# B&R Automation Studio project TD52 (part 95)

#### VibMonEGInit.st
```iecst
(*******************************************************************************
VibMonEG: Vigration monitoring engine / generator (init)

This code is confidential AND proprietary to the INNIO Company.
It may NOT be used in any form, or reproduced in any manner, without the express
written permission of the INNIO Company.
Copyright, INNIO Company, 2021

- monitoring of vibration values incl. frequency bands
- determine max velocity and frequencay at maximum

Customized modifications: -
------------------------

History:
-------
V4.11.0	25-05-2021	Weitzer, 	generated
V4.11.1	04-02-2022	Schmid,		automatic PLC address detection
V4.11.2	20-01-2026	Bacci,		customized for DP29

Instructions FOR use:
--------------------
Sensor 1: Generator horizontal
Sensor 2: Generator vetical
Sensor 3: Engine horizontal
Sensor 4: Engine vetical

Outstandings:
------------

*******************************************************************************)

PROGRAM _INIT

//	(*========= DETERMINE POSITION OF X20CM4810 MODULE ==========*)
//	(* ********************************************************* *)
//	(*	reset variables											 *)
//	(* ********************************************************* *)
//	memset(ADR(sLabelInfo),	 	0, SIZEOF(sLabelInfo));
//
//	(* ********************************************************* *)
//	(*	get information about configured modules				 *)
//	(* ********************************************************* *)
//	xDiagCreateInfo_CM4810.enable	:= TRUE;
//	xDiagCreateInfo_CM4810.infoKind	:= asdiagCONFIGURED;
//	xDiagCreateInfo_CM4810();
//
//	IF (xDiagCreateInfo_CM4810.status = 0) THEN
//		iIdent 		:= xDiagCreateInfo_CM4810.ident;
//		iNrEntries	:= xDiagCreateInfo_CM4810.nrEntries;
//	END_IF;
//
//	(* ********************************************************* *)
//	(*	get module type of configured modules in Physical		 *)
//	(* ********************************************************* *)
//	FOR iIndex := 0 TO iNrEntries - 1 DO
//		xDiagGetStrInfo_CM4810.enable		:= TRUE;
//		xDiagGetStrInfo_CM4810.ident		:= iIdent;
//		xDiagGetStrInfo_CM4810.index		:= iIndex;
//		xDiagGetStrInfo_CM4810.infoCode		:= asdiagCONFIG_MODULE;
//		xDiagGetStrInfo_CM4810.pBuffer		:= ADR(sLabelInfo);
//		xDiagGetStrInfo_CM4810.bufferLen	:= SIZEOF(sLabelInfo) - 1;
//		xDiagGetStrInfo_CM4810();
//
//		IF (xDiagGetStrInfo_CM4810.status = 0) THEN
//		(* ********************************************************* *)
//		(*	get path of X20CM4810 module							 *)
//		(* ********************************************************* *)
//			IF FIND(sLabelInfo, 'X20CM4810') <> 0 THEN
//				xDiagGetStrInfo_CM4810.infoCode		:= asdiagPATH;
//				xDiagGetStrInfo_CM4810.pBuffer		:= ADR(sAddrInfo);
//				xDiagGetStrInfo_CM4810.bufferLen	:= SIZEOF(sAddrInfo) - 1;
//				xDiagGetStrInfo_CM4810();
//
//				IF (xDiagGetStrInfo_CM4810.status = 0) THEN
//					sCM4810Addr	:=	sAddrInfo;
//				END_IF;
//			END_IF;
//		END_IF;
//	END_FOR;
//
//	(* ********************************************************* *)
//	(*	free ressources of AsIODiag								 *)
//	(* ********************************************************* *)
//	xDiagDisposeInfo_CM4810.enable := TRUE;
//	xDiagDisposeInfo_CM4810.ident  := iIdent;
//	xDiagDisposeInfo_CM4810();
//	(*===========================================================*)

//  Prevent compiler warnings
	xDiagCreateInfo_CM4810.enable := FALSE;
	xDiagGetStrInfo_CM4810.enable := FALSE;
	xDiagDisposeInfo_CM4810.enable := FALSE;
	sLabelInfo;
	sAddrInfo;
	iIndex;
	iIdent;
	iNrEntries;

	//  PLC address of 1st X20CM4810 vibration module
	sCM4810Addr := 'IF3.ST33.IF1.ST2';

	(* init setting for CM4810 FUB *)
	xCM4810.paramMain.pModulePath			  := ADR(sCM4810Addr); 								(* set path to module *)

	xCM4810.enable							  := TRUE; 											(* enable FUB *)
	xCM4810.paramBufferUpload.nrArrayElements := SIZEOF(rData_x_Axis)/SIZEOF(rData_x_Axis[0]);	(* the length of the rData_x_Axis and rData_y_Axis arrays must be the same *)
	xCM4810.paramBufferUpload.pArrayXaxis	  := ADR(rData_x_Axis);								(* load buffer address x axis array *)
	xCM4810.paramBufferUpload.pArrayYaxis	  := ADR(rData_y_Axis);								(* load buffer address y axis array *)

	xCM4810.paramBufferUpload.moduleBuffer:= 66;    (* define module buffer for upload *)
	//moduleBuffer  Buffer description                        Signal source             Channel number   Number of values   y-axis unit    x-axis unit
	//    9         Buffered time signal (amplitude)          Raw acceleration signal      1                8192                [mg]       [seconds]
	//   11         Buffered time signal (amplitude)          Raw acceleration signal      2                8192                [mg]       [seconds]
	//   13         Buffered time signal (amplitude)          Raw acceleration signal      3                8192                [mg]       [seconds]
	//   15         Buffered time signal (amplitude)          Raw acceleration signal      4                8192                [mg]       [seconds]
	//   25         Buffered time signal (amplitude)          Envelope monitoring          1                8192                [mg]       [seconds]
	//   27         Buffered time signal (amplitude)          Envelope monitoring          2                8192                [mg]       [seconds]
	//   29         Buffered time signal (amplitude)          Envelope monitoring          3                8192                [mg]       [seconds]
	//   31         Buffered time signal (amplitude)          Envelope monitoring          4                8192                [mg]       [seconds]
	//   66         Spectrum buffered frequency (amplitude)   Raw velocity signal          1                4096                [mm/s]       [Hz]
	//   67         Spectrum buffered frequency (amplitude)   Raw acceleration signal      1                4096                [mg]         [Hz]
	//   70         Spectrum buffered frequency (amplitude)   Raw velocity signal          2                4096                [mm/s]       [Hz]
	//   71         Spectrum buffered frequency (amplitude)   Raw acceleration signal      2                4096                [mg]         [Hz]
	//   74         Spectrum buffered frequency (amplitude)   Raw velocity signal          3                4096                [mm/s]       [Hz]
	//   75         Spectrum buffered frequency (amplitude)   Raw acceleration signal      3                4096                [mg]         [Hz]
	//   78         Spectrum buffered frequency (amplitude)   Raw velocity signal          4                4096                [mm/s]       [Hz]
	//   79         Spectrum buffered frequency (amplitude)   Raw acceleration signal      4                4096                [mg]         [Hz]
	//   82         Spectrum buffered frequency (amplitude)   Envelope signal speed        1                4096                [mm/s]       [Hz]
	//   83         Spectrum buffered frequency (amplitude)   Envelope monitoring          1                4096                [mg]         [Hz]
	//   86         Spectrum buffered frequency (amplitude)   Envelope signal speed        2                4096                [mm/s]       [Hz]
	//   87         Spectrum buffered frequency (amplitude)   Envelope monitoring          2                4096                [mg]         [Hz]
	//   90         Spectrum buffered frequency (amplitude)   Envelope signal speed        3                4096                [mm/s]       [Hz]
	//   91         Spectrum buffered frequency (amplitude)   Envelope monitoring          3                4096                [mg]         [Hz]
	//   94         Spectrum buffered frequency (amplitude)   Envelope signal speed        4                4096                [mm/s]       [Hz]
	//   95         Spectrum buffered frequency (amplitude)   Envelope monitoring          4                4096                [mg]         [Hz]

	(* set sensor sensitivity *)
	rSensitivitySensor[1] := 100.0; (*mV/g*)
	rSensitivitySensor[2] := 100.0; (*mV/g*)
	rSensitivitySensor[3] := 100.0; (*mV/g*)
	rSensitivitySensor[4] := 100.0; (*mV/g*)

	(* Enable application of sensitivity on buffer *)
	xCM4810.paramMain.sensitivitySensor01:=rSensitivitySensor[1];
	xCM4810.paramMain.sensitivitySensor02:=rSensitivitySensor[2];
	xCM4810.paramMain.sensitivitySensor03:=rSensitivitySensor[3];
	xCM4810.paramMain.sensitivitySensor04:=rSensitivitySensor[4];

	(* initialize values *)
	tiCM4810_ReadBuffer := T#1m;
	iNum_VibSens		:= 1;

END_PROGRAM
```

#### VibMonEG.typ - Local data types
```iecst
TYPE
	stpCM4810_Enum :
		(
		stpInitDone,
		stpWaitStart,
		stpReqLockBuffer,
		stpUploadBuffer,
		stpReqUnlockBuffer,
		stpError
		);
END_TYPE
```

#### VibMonEG.var - Local variables
```iecst
VAR CONSTANT
	AxisArrayMaxIndex : UINT := 8191;
END_VAR
VAR
	bStartBufferUpload : BOOL := TRUE; (* in order to start the buffer upload, set to TRUE *)
	xCM4810 : vbioCtrlCM4810; (* FUB to read buffers of a CM4810 module *)
	stpCM4810 : stpCM4810_Enum; (* step of state machine *)
	rData_x_Axis : ARRAY[0..AxisArrayMaxIndex] OF REAL; (* array of x-axis values (time values [s] or frequency values [Hz]) *)
	rData_y_Axis : ARRAY[0..AxisArrayMaxIndex] OF REAL; (* array of y-axis values (vibration [mg] of [mm/s] values *)
	bWrite : BOOL;
	szWriteConfig : STRING[50];
	bRead : BOOL;
	szReadConfig : STRING[50];
	xAsIOAccWrite1 : AsIOAccWrite;
	xAsIOAccRead1 : AsIOAccRead;
	rSensitivitySensor : ARRAY[0..4] OF REAL;
	bGetFrequencyMax : BOOL;
	usCount : UINT;
	tiCM4810_ReadBuffer : TIME;
	xTON_ReadCycle : TON;
	iNum_VibSens : INT;
	rVel_VibSens_Band : ARRAY[0..32] OF REAL := [33(0)];
	rVel_VibSens : ARRAY[0..4] OF REAL := [5(0)];
	usMaxIndex : UINT;
	rVel_y_Axis_Max : REAL;
	bVibSens_Overflow : ARRAY[0..4] OF BOOL := [5(0)];
	bVibSens_BrokenWire : ARRAY[0..4] OF BOOL := [5(0)];
	ucWriteBandCnt : USINT := 0;
	rCenterBandOld1 : REAL := 0.0;
	rCenterBandOld2 : REAL := 0.0;
	rCenterBandOld3 : REAL := 0.0;
	rCenterBandOld4 : REAL := 0.0;
	rCenterBandOld5 : REAL := 0.0;
	rCenterBandOld6 : REAL := 0.0;
	rCenterBandOld7 : REAL := 0.0;
	rCenterBandOld8 : REAL := 0.0;
	rIdx_VibSens_BandWidtOld : REAL := 0.0;
END_VAR
VAR
	xDiagCreateInfo_CM4810 : DiagCreateInfo; (*Get number of configured modules*)
	xDiagGetStrInfo_CM4810 : DiagGetStrInfo; (*Get name of configured modules*)
	xDiagDisposeInfo_CM4810 : DiagDisposeInfo; (*Free ressources of AsIODiag*)
	sLabelInfo : STRING[50]; (*Includes label of configured module*)
	sAddrInfo : STRING[50]; (*Includes address of configured module*)
	iIndex : UDINT; (*Index of actual read module*)
	iIdent : UDINT; (*Ident from xDiagCreateInfo_CM4810*)
	iNrEntries : UDINT; (*Number of configured modules from xDiagCreateInfo_CM4810*)
	sCM4810Addr : STRING[50]; (*CM4810 IF PLC address string*)
END_VAR
```

### Program Logical/EngineGeneral/VibMon2EG (IEC, version 4.11.1) - Vibration monitoring eng & gen

#### VibMonEGCyclic.st - Init, cyclic, exit code
```iecst
(*******************************************************************************
VibMonEG: Vigration monitoring engine / generator (cyclic)

This code is confidential AND proprietary to the INNIO Company.
It may NOT be used in any form, or reproduced in any manner, without the express
written permission of the INNIO Company.
Copyright, INNIO Company, 2021

- monitoring of vibration values incl. frequency bands
- determine max velocity and frequencay at maximum

Customized modifications: -
------------------------

History:
-------
V4.11	25-05-2021	Weitzer, 	generated

Instructions FOR use:
--------------------
Sensor 1: Generator horizontal
Sensor 2: Generator vetical
Sensor 3: Engine horizontal
Sensor 4: Engine vetical

Outstandings:
------------

*******************************************************************************)

PROGRAM _CYCLIC

	(* code is only executed if function is activated by parameter and if system has completed the start up *)
	IF Para.bVibSens_Act AND IN_EG.tPB2MM.bSys_Run THEN

		(* mapping of data points from 4 vibration sensors *)
		FOR usCount := 0 TO 3 DO

			(* check if vibraton sensore wire break detected and engine speed is below start limit *)
			IF bVibSens_BrokenWire[usCount+1] OR IN_EG.rN_EngAct < Para.rN_EngStart_LimHi THEN
				(* vibration sensor live RMS values [mm/s]*)
				MM2VIS.rVel_VibSens[usCount+5] := 0;
				(* vibration sensor live frequency band [mm/s] *)
				MM2VIS.rVel_VibSens_Band1[usCount+5] := 0;
				MM2VIS.rVel_VibSens_Band2[usCount+5] := 0;
				MM2VIS.rVel_VibSens_Band3[usCount+5] := 0;
				MM2VIS.rVel_VibSens_Band4[usCount+5] := 0;
				MM2VIS.rVel_VibSens_Band5[usCount+5] := 0;
				MM2VIS.rVel_VibSens_Band6[usCount+5] := 0;
				MM2VIS.rVel_VibSens_Band7[usCount+5] := 0;
				MM2VIS.rVel_VibSens_Band8[usCount+5] := 0;
				(* vibration sensor max values *)
				MM2VIS.rVel_VibSens_Max[usCount+5] := 0;
				MM2VIS.rF_VibSens_Max[usCount+5]   := 0;
			(* check if no vibraton sensore overflow detected *)
			ELSIF NOT bVibSens_Overflow[usCount+1] THEN
				(* vibration sensor live RMS values [mm/s]*)
				MM2VIS.rVel_VibSens[usCount+5] := rVel_VibSens[usCount+1];					(* mapping directly from IO mapping, no HALIO used for vibration mesarurement *)
				(* vibration sensor live frequency band [mm/s] *)
				MM2VIS.rVel_VibSens_Band1[usCount+5] := rVel_VibSens_Band[usCount*8+1];		(* mapping directly from IO mapping, no HALIO used for vibration mesarurement *)
				MM2VIS.rVel_VibSens_Band2[usCount+5] := rVel_VibSens_Band[usCount*8+2];		(* mapping directly from IO mapping, no HALIO used for vibration mesarurement *)
				MM2VIS.rVel_VibSens_Band3[usCount+5] := rVel_VibSens_Band[usCount*8+3];		(* mapping directly from IO mapping, no HALIO used for vibration mesarurement *)
				MM2VIS.rVel_VibSens_Band4[usCount+5] := rVel_VibSens_Band[usCount*8+4];		(* mapping directly from IO mapping, no HALIO used for vibration mesarurement *)
				MM2VIS.rVel_VibSens_Band5[usCount+5] := rVel_VibSens_Band[usCount*8+5];		(* mapping directly from IO mapping, no HALIO used for vibration mesarurement *)
				MM2VIS.rVel_VibSens_Band6[usCount+5] := rVel_VibSens_Band[usCount*8+6];		(* mapping directly from IO mapping, no HALIO used for vibration mesarurement *)
				MM2VIS.rVel_VibSens_Band7[usCount+5] := rVel_VibSens_Band[usCount*8+7];		(* mapping directly from IO mapping, no HALIO used for vibration mesarurement *)
				MM2VIS.rVel_VibSens_Band8[usCount+5] := rVel_VibSens_Band[usCount*8+8];		(* mapping directly from IO mapping, no HALIO used for vibration mesarurement *)
			END_IF;

		END_FOR;

		(* read buffer data *)

		(* generate time interval for reading buffer *)
		xTON_ReadCycle(IN := NOT xTON_ReadCycle.Q, PT :=  tiCM4810_ReadBuffer);

		(* generate start reading trigger *)
		IF IN_EG.tEng_Run.Do AND stpCM4810 = stpWaitStart AND xTON_ReadCycle.Q THEN
			iNum_VibSens := iNum_VibSens + 1;
			IF iNum_VibSens > 4 THEN
				iNum_VibSens := 1;
			END_IF;
			bStartBufferUpload 					   := TRUE;
			xCM4810.paramBufferUpload.moduleBuffer := 66 + (iNum_VibSens-1) * 4;
		END_IF;

		(* state engine to read of data buffer *)

		CASE stpCM4810 OF
			//---------------------------------------------
			// wait for init done
			//---------------------------------------------
			stpInitDone:
				xCM4810.requestBufferLock := FALSE;
				xCM4810.uploadBuffer	  := FALSE;
				IF xCM4810.initDone AND xCM4810.moduleCfgUploadDone THEN
					stpCM4810 := stpWaitStart;
				END_IF;

			//---------------------------------------------
			// wait for start uplaod buffer
			//---------------------------------------------
			stpWaitStart:
				xCM4810.requestBufferLock := FALSE;
				xCM4810.uploadBuffer	  := FALSE;
				(* wait for start *)
				IF bStartBufferUpload THEN
					stpCM4810 := stpReqLockBuffer;
				END_IF;

			//---------------------------------------------
			// request lock buffer and wait until valid
			//---------------------------------------------
			stpReqLockBuffer:
				xCM4810.requestBufferLock := TRUE;
				bStartBufferUpload		  := FALSE; (* reset command start *)
				IF xCM4810.bufferLockValid THEN
					xCM4810.uploadBuffer := TRUE;
					stpCM4810			 := stpUploadBuffer;
				END_IF;

			//---------------------------------------------
			// upload buffer
			//---------------------------------------------
			stpUploadBuffer:
				IF xCM4810.bufferUploadDone THEN
					stpCM4810 := stpReqUnlockBuffer;
				END_IF;
				IF xCM4810.status <> ERR_FUB_BUSY AND xCM4810.status <> ERR_OK THEN
					stpCM4810 := stpError;
				END_IF

			//---------------------------------------------
			// unlock buffer and wait until valid
			//---------------------------------------------
			stpReqUnlockBuffer:
				xCM4810.requestBufferLock := FALSE;
				xCM4810.uploadBuffer	  := FALSE;
				IF NOT xCM4810.bufferLockValid THEN
					bGetFrequencyMax := TRUE;
					stpCM4810		 := stpWaitStart;
				END_IF;

			//---------------------------------------------
			// error
			//---------------------------------------------
			stpError:
			// no action!

		END_CASE;

		xCM4810.paramMain.pModulePath			  := ADR(sCM4810Addr);
		xCM4810.paramBufferUpload.pArrayXaxis	  := ADR(rData_x_Axis);
		xCM4810.paramBufferUpload.pArrayYaxis	  := ADR(rData_y_Axis);

		xCM4810(); (* call FUB exactly once per cycle *)

		(* get value & frequency max *)

		IF bGetFrequencyMax THEN

			MM2VIS.rF_VibSens_Max[iNum_VibSens+4]   := 0.0;		(* reset x(y max) max *)
			rVel_y_Axis_Max := 0.0;										(* reset y max *)
			usMaxIndex := 0;
			FOR usCount := 1 TO AxisArrayMaxIndex DO
				(* Upper limit for max value search at 500 Hz *)
				IF rData_x_Axis[usCount] > 500.0 THEN
					EXIT;
				END_IF
				(*find max signal value *)
				IF rData_y_Axis[usCount] > rVel_y_Axis_Max THEN
					rVel_y_Axis_Max := rData_y_Axis[usCount];		(* max virbration value *)
					MM2VIS.rF_VibSens_Max[iNum_VibSens+4]   := rData_x_Axis[usCount];		(* frequency at max virbration value *)
					usMaxIndex := usCount;
				END_IF
			END_FOR;

			(* correction of buffer value *)
			IF usMaxIndex > 1 AND usMaxIndex < (AxisArrayMaxIndex-2) THEN
				MM2VIS.rVel_VibSens_Max[iNum_VibSens+4] := 2.0/SQRT(3.0/2.0)*SQRT(0.5*(EXPT(rData_y_Axis[usMaxIndex-2],2)+EXPT(rData_y_Axis[usMaxIndex-1],2)+EXPT(rData_y_Axis[usMaxIndex],2)+EXPT(rData_y_Axis[usMaxIndex+1],2)+EXPT(rData_y_Axis[usMaxIndex+2],2)));
			ELSE
				MM2VIS.rVel_VibSens_Max[iNum_VibSens+4] := 0.0;
			END_IF;

			bGetFrequencyMax := FALSE;
		END_IF;

		(* calculate and display center frequency at the HMI *)

//		MM2VIS.rF_VibSens_CenterBand1 := Para.rN_EngNom/60.0*Para.rIdx_VibSens_BandOrder1;
//		MM2VIS.rF_VibSens_CenterBand2 := Para.rN_EngNom/60.0*Para.rIdx_VibSens_BandOrder2;
//		MM2VIS.rF_VibSens_CenterBand3 := Para.rN_EngNom/60.0*Para.rIdx_VibSens_BandOrder3;
//		MM2VIS.rF_VibSens_CenterBand4 := Para.rN_EngNom/60.0*Para.rIdx_VibSens_BandOrder4;
//		MM2VIS.rF_VibSens_CenterBand5 := Para.rN_EngNom/60.0*Para.rIdx_VibSens_BandOrder5;
//		MM2VIS.rF_VibSens_CenterBand6 := Para.rN_EngNom/60.0*Para.rIdx_VibSens_BandOrder6;
//		MM2VIS.rF_VibSens_CenterBand7 := Para.rN_EngNom/60.0*Para.rIdx_VibSens_BandOrder7;
//		MM2VIS.rF_VibSens_CenterBand8 := Para.rN_EngNom/60.0*Para.rIdx_VibSens_BandOrder8;

		(* check if band upper and lower frequency limit has to be set *)

		IF NOT bWrite THEN

			IF ucWriteBandCnt = 0 THEN

				IF Para.rIdx_VibSens_BandWidth <> rIdx_VibSens_BandWidtOld THEN
					rIdx_VibSens_BandWidtOld := Para.rIdx_VibSens_BandWidth;
					rCenterBandOld1			 := 0.0;
					rCenterBandOld2			 := 0.0;
					rCenterBandOld3			 := 0.0;
					rCenterBandOld4			 := 0.0;
					rCenterBandOld5			 := 0.0;
					rCenterBandOld6			 := 0.0;
					rCenterBandOld7			 := 0.0;
					rCenterBandOld8			 := 0.0;
				ELSIF MM2VIS.rF_VibSens_CenterBand1 <> rCenterBandOld1 THEN
					rCenterBandOld1 := MM2VIS.rF_VibSens_CenterBand1;
					ucWriteBandCnt  := 1;
				ELSIF MM2VIS.rF_VibSens_CenterBand2 <> rCenterBandOld2 THEN
					rCenterBandOld2 := MM2VIS.rF_VibSens_CenterBand2;
					ucWriteBandCnt  := 9;
				ELSIF MM2VIS.rF_VibSens_CenterBand3 <> rCenterBandOld3 THEN
					rCenterBandOld3 := MM2VIS.rF_VibSens_CenterBand3;
					ucWriteBandCnt  := 17;
				ELSIF MM2VIS.rF_VibSens_CenterBand4 <> rCenterBandOld4 THEN
					rCenterBandOld4 := MM2VIS.rF_VibSens_CenterBand4;
					ucWriteBandCnt  := 25;
				ELSIF MM2VIS.rF_VibSens_CenterBand5 <> rCenterBandOld5 THEN
					rCenterBandOld5 := MM2VIS.rF_VibSens_CenterBand5;
					ucWriteBandCnt  := 33;
				ELSIF MM2VIS.rF_VibSens_CenterBand6 <> rCenterBandOld6 THEN
					rCenterBandOld6 := MM2VIS.rF_VibSens_CenterBand6;
					ucWriteBandCnt  := 41;
				ELSIF MM2VIS.rF_VibSens_CenterBand7 <> rCenterBandOld7 THEN
					rCenterBandOld7 := MM2VIS.rF_VibSens_CenterBand7;
					ucWriteBandCnt  := 49;
				ELSIF MM2VIS.rF_VibSens_CenterBand8 <> rCenterBandOld8 THEN
					rCenterBandOld8 := MM2VIS.rF_VibSens_CenterBand8;
					ucWriteBandCnt  := 57;
				END_IF;

			END_IF;

			(* writing of the single band limit registers *)
			CASE ucWriteBandCnt OF

				(* Band 1 - Sensor 1 *)
				1:  bWrite		 		 := TRUE;
					szWriteConfig		 := 'FrequencyBand01LowerFrequency';
					xAsIOAccWrite1.value := LIMIT(1,REAL_TO_UDINT(4.0*(MM2VIS.rF_VibSens_CenterBand1 - Para.rIdx_VibSens_BandWidth/2)),40000);
					ucWriteBandCnt		 := 2;
				2:  bWrite		 		 := TRUE;
					szWriteConfig		 := 'FrequencyBand01UpperFrequency';
					xAsIOAccWrite1.value := LIMIT(1,REAL_TO_UDINT(4.0*(MM2VIS.rF_VibSens_CenterBand1 + Para.rIdx_VibSens_BandWidth/2)),40000);
					ucWriteBandCnt		 := 3;
				(* Band 1 - Sensor 2 *)
				3:  bWrite		 		 := TRUE;
					szWriteConfig		 := 'FrequencyBand09LowerFrequency';
					xAsIOAccWrite1.value := LIMIT(1,REAL_TO_UDINT(4.0*(MM2VIS.rF_VibSens_CenterBand1 - Para.rIdx_VibSens_BandWidth/2)),40000);
					ucWriteBandCnt		 := 4;
				4:  bWrite		 		 := TRUE;
					szWriteConfig		 := 'FrequencyBand09UpperFrequency';
					xAsIOAccWrite1.value := LIMIT(1,REAL_TO_UDINT(4.0*(MM2VIS.rF_VibSens_CenterBand1 + Para.rIdx_VibSens_BandWidth/2)),40000);
					ucWriteBandCnt		 := 5;
				(* Band 1 - Sensor 3 *)
				5:  bWrite		 		 := TRUE;
					szWriteConfig		 := 'FrequencyBand17LowerFrequency';
					xAsIOAccWrite1.value := LIMIT(1,REAL_TO_UDINT(4.0*(MM2VIS.rF_VibSens_CenterBand1 - Para.rIdx_VibSens_BandWidth/2)),40000);
					ucWriteBandCnt		 := 6;
				6:  bWrite		 		 := TRUE;
					szWriteConfig		 := 'FrequencyBand17UpperFrequency';
					xAsIOAccWrite1.value := LIMIT(1,REAL_TO_UDINT(4.0*(MM2VIS.rF_VibSens_CenterBand1 + Para.rIdx_VibSens_BandWidth/2)),40000);
					ucWriteBandCnt		 := 7;
				(* Band 1 - Sensor 4 *)
				7:  bWrite		 		 := TRUE;
					szWriteConfig		 := 'FrequencyBand25LowerFrequency';
					xAsIOAccWrite1.value := LIMIT(1,REAL_TO_UDINT(4.0*(MM2VIS.rF_VibSens_CenterBand1 - Para.rIdx_VibSens_BandWidth/2)),40000);
					ucWriteBandCnt		 := 8;
				8:  bWrite		 		 := TRUE;
					szWriteConfig		 := 'FrequencyBand25UpperFrequency';
					xAsIOAccWrite1.value := LIMIT(1,REAL_TO_UDINT(4.0*(MM2VIS.rF_VibSens_CenterBand1 + Para.rIdx_VibSens_BandWidth/2)),40000);
					ucWriteBandCnt		 := 0;

					(* Band 2 - Sensor 1 *)
				9:  bWrite		 		 := TRUE;
					szWriteConfig		 := 'FrequencyBand02LowerFrequency';
					xAsIOAccWrite1.value := LIMIT(1,REAL_TO_UDINT(4.0*(MM2VIS.rF_VibSens_CenterBand2 - Para.rIdx_VibSens_BandWidth/2)),40000);
					ucWriteBandCnt		 := 10;
				10: bWrite		 		 := TRUE;
					szWriteConfig		 := 'FrequencyBand02UpperFrequency';
					xAsIOAccWrite1.value := LIMIT(1,REAL_TO_UDINT(4.0*(MM2VIS.rF_VibSens_CenterBand2 + Para.rIdx_VibSens_BandWidth/2)),40000);
					ucWriteBandCnt		 := 11;
					(* Band 2 - Sensor 2 *)
				11: bWrite		 		 := TRUE;
					szWriteConfig		 := 'FrequencyBand10LowerFrequency';
					xAsIOAccWrite1.value := LIMIT(1,REAL_TO_UDINT(4.0*(MM2VIS.rF_VibSens_CenterBand2 - Para.rIdx_VibSens_BandWidth/2)),40000);
					ucWriteBandCnt		 := 12;
				12: bWrite		 		 := TRUE;
					szWriteConfig		 := 'FrequencyBand10UpperFrequency';
					xAsIOAccWrite1.value := LIMIT(1,REAL_TO_UDINT(4.0*(MM2VIS.rF_VibSens_CenterBand2 + Para.rIdx_VibSens_BandWidth/2)),40000);
					ucWriteBandCnt		 := 13;
					(* Band 2 - Sensor 3 *)
				13: bWrite		 		 := TRUE;
					szWriteConfig		 := 'FrequencyBand18LowerFrequency';
					xAsIOAccWrite1.value := LIMIT(1,REAL_TO_UDINT(4.0*(MM2VIS.rF_VibSens_CenterBand2 - Para.rIdx_VibSens_BandWidth/2)),40000);
					ucWriteBandCnt		 := 14;
				14: bWrite		 		 := TRUE;
					szWriteConfig		 := 'FrequencyBand18UpperFrequency';
					xAsIOAccWrite1.value := LIMIT(1,REAL_TO_UDINT(4.0*(MM2VIS.rF_VibSens_CenterBand2 + Para.rIdx_VibSens_BandWidth/2)),40000);
					ucWriteBandCnt		 := 15;
					(* Band 2 - Sensor 4 *)
				15: bWrite		 		 := TRUE;
					szWriteConfig		 := 'FrequencyBand26LowerFrequency';
					xAsIOAccWrite1.value := LIMIT(1,REAL_TO_UDINT(4.0*(MM2VIS.rF_VibSens_CenterBand2 - Para.rIdx_VibSens_BandWidth/2)),40000);
					ucWriteBandCnt		 := 16;
				16: bWrite		 		 := TRUE;
					szWriteConfig		 := 'FrequencyBand26UpperFrequency';
					xAsIOAccWrite1.value := LIMIT(1,REAL_TO_UDINT(4.0*(MM2VIS.rF_VibSens_CenterBand2 + Para.rIdx_VibSens_BandWidth/2)),40000);
					ucWriteBandCnt		 := 0;

					(* Band 3 - Sensor 1 *)
				17: bWrite		 		 := TRUE;
					szWriteConfig		 := 'FrequencyBand03LowerFrequency';
					xAsIOAccWrite1.value := LIMIT(1,REAL_TO_UDINT(4.0*(MM2VIS.rF_VibSens_CenterBand3 - Para.rIdx_VibSens_BandWidth/2)),40000);
					ucWriteBandCnt		 := 18;
				18: bWrite		 		 := TRUE;
					szWriteConfig		 := 'FrequencyBand03UpperFrequency';
					xAsIOAccWrite1.value := LIMIT(1,REAL_TO_UDINT(4.0*(MM2VIS.rF_VibSens_CenterBand3 + Para.rIdx_VibSens_BandWidth/2)),40000);
					ucWriteBandCnt		 := 19;
					(* Band 3 - Sensor 2 *)
				19: bWrite		 		 := TRUE;
					szWriteConfig		 := 'FrequencyBand11LowerFrequency';
					xAsIOAccWrite1.value := LIMIT(1,REAL_TO_UDINT(4.0*(MM2VIS.rF_VibSens_CenterBand3 - Para.rIdx_VibSens_BandWidth/2)),40000);
					ucWriteBandCnt		 := 20;
				20: bWrite		 		 := TRUE;
					szWriteConfig		 := 'FrequencyBand11UpperFrequency';
					xAsIOAccWrite1.value := LIMIT(1,REAL_TO_UDINT(4.0*(MM2VIS.rF_VibSens_CenterBand3 + Para.rIdx_VibSens_BandWidth/2)),40000);
					ucWriteBandCnt		 := 21;
					(* Band 3 - Sensor 3 *)
				21: bWrite		 		 := TRUE;
					szWriteConfig		 := 'FrequencyBand19LowerFrequency';
					xAsIOAccWrite1.value := LIMIT(1,REAL_TO_UDINT(4.0*(MM2VIS.rF_VibSens_CenterBand3 - Para.rIdx_VibSens_BandWidth/2)),40000);
					ucWriteBandCnt		 := 22;
				22: bWrite		 		 := TRUE;
					szWriteConfig		 := 'FrequencyBand19UpperFrequency';
					xAsIOAccWrite1.value := LIMIT(1,REAL_TO_UDINT(4.0*(MM2VIS.rF_VibSens_CenterBand3 + Para.rIdx_VibSens_BandWidth/2)),40000);
					ucWriteBandCnt		 := 23;
					(* Band 3 - Sensor 4 *)
				23: bWrite		 		 := TRUE;
					szWriteConfig		 := 'FrequencyBand27LowerFrequency';
					xAsIOAccWrite1.value := LIMIT(1,REAL_TO_UDINT(4.0*(MM2VIS.rF_VibSens_CenterBand3 - Para.rIdx_VibSens_BandWidth/2)),40000);
					ucWriteBandCnt		 := 24;
				24: bWrite		 		 := TRUE;
					szWriteConfig		 := 'FrequencyBand27UpperFrequency';
					xAsIOAccWrite1.value := LIMIT(1,REAL_TO_UDINT(4.0*(MM2VIS.rF_VibSens_CenterBand3 + Para.rIdx_VibSens_BandWidth/2)),40000);
					ucWriteBandCnt		 := 0;

					(* Band 4 - Sensor 1 *)
				25: bWrite		 		 := TRUE;
					szWriteConfig		 := 'FrequencyBand04LowerFrequency';
					xAsIOAccWrite1.value := LIMIT(1,REAL_TO_UDINT(4.0*(MM2VIS.rF_VibSens_CenterBand4 - Para.rIdx_VibSens_BandWidth/2)),40000);
					ucWriteBandCnt		 := 26;
				26: bWrite		 		 := TRUE;
					szWriteConfig		 := 'FrequencyBand04UpperFrequency';
					xAsIOAccWrite1.value := LIMIT(1,REAL_TO_UDINT(4.0*(MM2VIS.rF_VibSens_CenterBand4 + Para.rIdx_VibSens_BandWidth/2)),40000);
					ucWriteBandCnt		 := 27;
					(* Band 4 - Sensor 2 *)
				27: bWrite		 		 := TRUE;
					szWriteConfig		 := 'FrequencyBand12LowerFrequency';
					xAsIOAccWrite1.value := LIMIT(1,REAL_TO_UDINT(4.0*(MM2VIS.rF_VibSens_CenterBand4 - Para.rIdx_VibSens_BandWidth/2)),40000);
					ucWriteBandCnt		 := 28;
				28: bWrite		 		 := TRUE;
					szWriteConfig		 := 'FrequencyBand12UpperFrequency';
					xAsIOAccWrite1.value := LIMIT(1,REAL_TO_UDINT(4.0*(MM2VIS.rF_VibSens_CenterBand4 + Para.rIdx_VibSens_BandWidth/2)),40000);
					ucWriteBandCnt		 := 29;
					(* Band 4 - Sensor 3 *)
				29: bWrite		 		 := TRUE;
					szWriteConfig		 := 'FrequencyBand20LowerFrequency';
					xAsIOAccWrite1.value := LIMIT(1,REAL_TO_UDINT(4.0*(MM2VIS.rF_VibSens_CenterBand4 - Para.rIdx_VibSens_BandWidth/2)),40000);
					ucWriteBandCnt		 := 30;
				30: bWrite		 		 := TRUE;
					szWriteConfig		 := 'FrequencyBand20UpperFrequency';
					xAsIOAccWrite1.value := LIMIT(1,REAL_TO_UDINT(4.0*(MM2VIS.rF_VibSens_CenterBand4 + Para.rIdx_VibSens_BandWidth/2)),40000);
					ucWriteBandCnt		 := 31;
					(* Band 4 - Sensor 4 *)
				31: bWrite		 		 := TRUE;
					szWriteConfig		 := 'FrequencyBand28LowerFrequency';
					xAsIOAccWrite1.value := LIMIT(1,REAL_TO_UDINT(4.0*(MM2VIS.rF_VibSens_CenterBand4 - Para.rIdx_VibSens_BandWidth/2)),40000);
					ucWriteBandCnt		 := 32;
				32: bWrite		 		 := TRUE;
					szWriteConfig		 := 'FrequencyBand28UpperFrequency';
					xAsIOAccWrite1.value := LIMIT(1,REAL_TO_UDINT(4.0*(MM2VIS.rF_VibSens_CenterBand4 + Para.rIdx_VibSens_BandWidth/2)),40000);
					ucWriteBandCnt		 := 0;

					(* Band 5 - Sensor 1 *)
				33: bWrite		 		 := TRUE;
					szWriteConfig		 := 'FrequencyBand05LowerFrequency';
					xAsIOAccWrite1.value := LIMIT(1,REAL_TO_UDINT(4.0*(MM2VIS.rF_VibSens_CenterBand5 - Para.rIdx_VibSens_BandWidth/2)),40000);
					ucWriteBandCnt		 := 34;
				34: bWrite		 		 := TRUE;
					szWriteConfig		 := 'FrequencyBand05UpperFrequency';
					xAsIOAccWrite1.value := LIMIT(1,REAL_TO_UDINT(4.0*(MM2VIS.rF_VibSens_CenterBand5 + Para.rIdx_VibSens_BandWidth/2)),40000);
					ucWriteBandCnt		 := 35;
					(* Band 5 - Sensor 2 *)
				35: bWrite		 		 := TRUE;
					szWriteConfig		 := 'FrequencyBand13LowerFrequency';
					xAsIOAccWrite1.value := LIMIT(1,REAL_TO_UDINT(4.0*(MM2VIS.rF_VibSens_CenterBand5 - Para.rIdx_VibSens_BandWidth/2)),40000);
					ucWriteBandCnt		 := 36;
				36: bWrite		 		 := TRUE;
					szWriteConfig		 := 'FrequencyBand13UpperFrequency';
					xAsIOAccWrite1.value := LIMIT(1,REAL_TO_UDINT(4.0*(MM2VIS.rF_VibSens_CenterBand5 + Para.rIdx_VibSens_BandWidth/2)),40000);
					ucWriteBandCnt		 := 37;
					(* Band 5 - Sensor 3 *)
				37: bWrite		 		 := TRUE;
					szWriteConfig		 := 'FrequencyBand21LowerFrequency';
					xAsIOAccWrite1.value := LIMIT(1,REAL_TO_UDINT(4.0*(MM2VIS.rF_VibSens_CenterBand5 - Para.rIdx_VibSens_BandWidth/2)),40000);
					ucWriteBandCnt		 := 38;
				38: bWrite		 		 := TRUE;
					szWriteConfig		 := 'FrequencyBand21UpperFrequency';
					xAsIOAccWrite1.value := LIMIT(1,REAL_TO_UDINT(4.0*(MM2VIS.rF_VibSens_CenterBand5 + Para.rIdx_VibSens_BandWidth/2)),40000);
					ucWriteBandCnt		 := 39;
					(* Band 5 - Sensor 4 *)
				39: bWrite		 		 := TRUE;
					szWriteConfig		 := 'FrequencyBand29LowerFrequency';
					xAsIOAccWrite1.value := LIMIT(1,REAL_TO_UDINT(4.0*(MM2VIS.rF_VibSens_CenterBand5 - Para.rIdx_VibSens_BandWidth/2)),40000);
					ucWriteBandCnt		 := 40;
				40: bWrite		 		 := TRUE;
					szWriteConfig		 := 'FrequencyBand29UpperFrequency';
					xAsIOAccWrite1.value := LIMIT(1,REAL_TO_UDINT(4.0*(MM2VIS.rF_VibSens_CenterBand5 + Para.rIdx_VibSens_BandWidth/2)),40000);
					ucWriteBandCnt		 := 0;

					(* Band 6 - Sensor 1 *)
				41: bWrite		 		 := TRUE;
					szWriteConfig		 := 'FrequencyBand06LowerFrequency';
					xAsIOAccWrite1.value := LIMIT(1,REAL_TO_UDINT(4.0*(MM2VIS.rF_VibSens_CenterBand6 - Para.rIdx_VibSens_BandWidth/2)),40000);
					ucWriteBandCnt		 := 42;
				42: bWrite		 		 := TRUE;
					szWriteConfig		 := 'FrequencyBand06UpperFrequency';
					xAsIOAccWrite1.value := LIMIT(1,REAL_TO_UDINT(4.0*(MM2VIS.rF_VibSens_CenterBand6 + Para.rIdx_VibSens_BandWidth/2)),40000);
					ucWriteBandCnt		 := 43;
					(* Band 6 - Sensor 2 *)
				43: bWrite		 		 := TRUE;
					szWriteConfig		 := 'FrequencyBand14LowerFrequency';
					xAsIOAccWrite1.value := LIMIT(1,REAL_TO_UDINT(4.0*(MM2VIS.rF_VibSens_CenterBand6 - Para.rIdx_VibSens_BandWidth/2)),40000);
					ucWriteBandCnt		 := 44;
				44: bWrite		 		 := TRUE;
					szWriteConfig		 := 'FrequencyBand14UpperFrequency';
					xAsIOAccWrite1.value := LIMIT(1,REAL_TO_UDINT(4.0*(MM2VIS.rF_VibSens_CenterBand6 + Para.rIdx_VibSens_BandWidth/2)),40000);
					ucWriteBandCnt		 := 45;
					(* Band 6 - Sensor 3 *)
				45: bWrite		 		 := TRUE;
					szWriteConfig		 := 'FrequencyBand22LowerFrequency';
					xAsIOAccWrite1.value := LIMIT(1,REAL_TO_UDINT(4.0*(MM2VIS.rF_VibSens_CenterBand6 - Para.rIdx_VibSens_BandWidth/2)),40000);
					ucWriteBandCnt		 := 46;
				46: bWrite		 		 := TRUE;
					szWriteConfig		 := 'FrequencyBand22UpperFrequency';
					xAsIOAccWrite1.value := LIMIT(1,REAL_TO_UDINT(4.0*(MM2VIS.rF_VibSens_CenterBand6 + Para.rIdx_VibSens_BandWidth/2)),40000);
					ucWriteBandCnt		 := 47;
					(* Band 6 - Sensor 4 *)
				47: bWrite		 		 := TRUE;
					szWriteConfig		 := 'FrequencyBand30LowerFrequency';
					xAsIOAccWrite1.value := LIMIT(1,REAL_TO_UDINT(4.0*(MM2VIS.rF_VibSens_CenterBand6 - Para.rIdx_VibSens_BandWidth/2)),40000);
					ucWriteBandCnt		 := 48;
				48: bWrite		 		 := TRUE;
					szWriteConfig		 := 'FrequencyBand30UpperFrequency';
					xAsIOAccWrite1.value := LIMIT(1,REAL_TO_UDINT(4.0*(MM2VIS.rF_VibSens_CenterBand6 + Para.rIdx_VibSens_BandWidth/2)),40000);
					ucWriteBandCnt		 := 0;

					(* Band 7 - Sensor 1 *)
				49: bWrite		 		 := TRUE;
					szWriteConfig		 := 'FrequencyBand07LowerFrequency';
					xAsIOAccWrite1.value := LIMIT(1,REAL_TO_UDINT(4.0*(MM2VIS.rF_VibSens_CenterBand7 - Para.rIdx_VibSens_BandWidth/2)),40000);
					ucWriteBandCnt		 := 50;
				50: bWrite		 		 := TRUE;
					szWriteConfig		 := 'FrequencyBand07UpperFrequency';
					xAsIOAccWrite1.value := LIMIT(1,REAL_TO_UDINT(4.0*(MM2VIS.rF_VibSens_CenterBand7 + Para.rIdx_VibSens_BandWidth/2)),40000);
					ucWriteBandCnt		 := 51;
					(* Band 7 - Sensor 2 *)
				51: bWrite		 		 := TRUE;
					szWriteConfig		 := 'FrequencyBand15LowerFrequency';
					xAsIOAccWrite1.value := LIMIT(1,REAL_TO_UDINT(4.0*(MM2VIS.rF_VibSens_CenterBand7 - Para.rIdx_VibSens_BandWidth/2)),40000);
					ucWriteBandCnt		 := 52;
				52: bWrite		 		 := TRUE;
					szWriteConfig		 := 'FrequencyBand15UpperFrequency';
					xAsIOAccWrite1.value := LIMIT(1,REAL_TO_UDINT(4.0*(MM2VIS.rF_VibSens_CenterBand7 + Para.rIdx_VibSens_BandWidth/2)),40000);
					ucWriteBandCnt		 := 53;
					(* Band 7 - Sensor 3 *)
				53: bWrite		 		 := TRUE;
					szWriteConfig		 := 'FrequencyBand23LowerFrequency';
					xAsIOAccWrite1.value := LIMIT(1,REAL_TO_UDINT(4.0*(MM2VIS.rF_VibSens_CenterBand7 - Para.rIdx_VibSens_BandWidth/2)),40000);
					ucWriteBandCnt		 := 54;
				54: bWrite		 		 := TRUE;
					szWriteConfig		 := 'FrequencyBand23UpperFrequency';
					xAsIOAccWrite1.value := LIMIT(1,REAL_TO_UDINT(4.0*(MM2VIS.rF_VibSens_CenterBand7 + Para.rIdx_VibSens_BandWidth/2)),40000);
					ucWriteBandCnt		 := 55;
					(* Band 7 - Sensor 4 *)
				55: bWrite		 		 := TRUE;
					szWriteConfig		 := 'FrequencyBand31LowerFrequency';
					xAsIOAccWrite1.value := LIMIT(1,REAL_TO_UDINT(4.0*(MM2VIS.rF_VibSens_CenterBand7 - Para.rIdx_VibSens_BandWidth/2)),40000);
					ucWriteBandCnt		 := 56;
				56: bWrite		 		 := TRUE;
					szWriteConfig		 := 'FrequencyBand31UpperFrequency';
					xAsIOAccWrite1.value := LIMIT(1,REAL_TO_UDINT(4.0*(MM2VIS.rF_VibSens_CenterBand7 + Para.rIdx_VibSens_BandWidth/2)),40000);
					ucWriteBandCnt		 := 0;

					(* Band 8 - Sensor 1 *)
				57: bWrite		 		 := TRUE;
					szWriteConfig		 := 'FrequencyBand08LowerFrequency';
					xAsIOAccWrite1.value := LIMIT(1,REAL_TO_UDINT(4.0*(MM2VIS.rF_VibSens_CenterBand8 - Para.rIdx_VibSens_BandWidth/2)),40000);
					ucWriteBandCnt		 := 58;
				58: bWrite		 		 := TRUE;
					szWriteConfig		 := 'FrequencyBand08UpperFrequency';
					xAsIOAccWrite1.value := LIMIT(1,REAL_TO_UDINT(4.0*(MM2VIS.rF_VibSens_CenterBand8 + Para.rIdx_VibSens_BandWidth/2)),40000);
					ucWriteBandCnt		 := 59;
					(* Band 8 - Sensor 2 *)
				59: bWrite		 		 := TRUE;
					szWriteConfig		 := 'FrequencyBand16LowerFrequency';
					xAsIOAccWrite1.value := LIMIT(1,REAL_TO_UDINT(4.0*(MM2VIS.rF_VibSens_CenterBand8 - Para.rIdx_VibSens_BandWidth/2)),40000);
					ucWriteBandCnt		 := 60;
				60: bWrite		 		 := TRUE;
					szWriteConfig		 := 'FrequencyBand16UpperFrequency';
					xAsIOAccWrite1.value := LIMIT(1,REAL_TO_UDINT(4.0*(MM2VIS.rF_VibSens_CenterBand8 + Para.rIdx_VibSens_BandWidth/2)),40000);
					ucWriteBandCnt		 := 61;
					(* Band 8 - Sensor 3 *)
				61: bWrite		 		 := TRUE;
					szWriteConfig		 := 'FrequencyBand24LowerFrequency';
					xAsIOAccWrite1.value := LIMIT(1,REAL_TO_UDINT(4.0*(MM2VIS.rF_VibSens_CenterBand8 - Para.rIdx_VibSens_BandWidth/2)),40000);
					ucWriteBandCnt		 := 62;
				62: bWrite		 		 := TRUE;
					szWriteConfig		 := 'FrequencyBand24UpperFrequency';
					xAsIOAccWrite1.value := LIMIT(1,REAL_TO_UDINT(4.0*(MM2VIS.rF_VibSens_CenterBand8 + Para.rIdx_VibSens_BandWidth/2)),40000);
					ucWriteBandCnt		 := 63;
					(* Band 8 - Sensor 4 *)
				63: bWrite		 		 := TRUE;
					szWriteConfig		 := 'FrequencyBand32LowerFrequency';
					xAsIOAccWrite1.value := LIMIT(1,REAL_TO_UDINT(4.0*(MM2VIS.rF_VibSens_CenterBand8 - Para.rIdx_VibSens_BandWidth/2)),40000);
					ucWriteBandCnt		 := 64;
				64: bWrite		 		 := TRUE;
					szWriteConfig		 := 'FrequencyBand32UpperFrequency';
					xAsIOAccWrite1.value := LIMIT(1,REAL_TO_UDINT(4.0*(MM2VIS.rF_VibSens_CenterBand8 + Para.rIdx_VibSens_BandWidth/2)),40000);
					ucWriteBandCnt		 := 0;

			END_CASE;

		END_IF;

		(* read & write X204810 registers *)

		(* write band configuration and miscellaneous values *)
		IF bWrite THEN														(* set bWrite to TRUE to write a register on the CM48810 X20 module *)
			xAsIOAccWrite1.enable	    := TRUE;
			xAsIOAccWrite1.pDeviceName  := xCM4810.paramMain.pModulePath;
//			xAsIOAccWrite1.value	    := 0;								(* set value to write at this attribute of the function block *)
			xAsIOAccWrite1.pChannelName	:= ADR(szWriteConfig);				(* set name of register to write at string pv szWriteConfig *)
			xAsIOAccWrite1();

			IF xAsIOAccWrite1.status = 0 THEN
				bWrite := FALSE;
			END_IF;
		END_IF;

		(* read miscellaneous values *)
		IF bRead THEN														(* set bRead to TRUE to read a register from the CM48810 X20 module *)
			xAsIOAccRead1.enable	   := TRUE;
			xAsIOAccRead1.pDeviceName  := xCM4810.paramMain.pModulePath;
//			xAsIOAccRead1.value;											(* here the read valure can be found *)
			xAsIOAccRead1.pChannelName := ADR(szReadConfig);				(* set name of register to read at string pv szReadConfig *)
			xAsIOAccRead1();

			IF xAsIOAccRead1.status = 0 THEN
				bRead := FALSE;
			END_IF;
		END_IF;

	END_IF;

END_PROGRAM
```

#### VibMonEGInit.st
```iecst
(*******************************************************************************
VibMonEG: Vigration monitoring engine / generator (init)

This code is confidential AND proprietary to the INNIO Company.
It may NOT be used in any form, or reproduced in any manner, without the express
written permission of the INNIO Company.
Copyright, INNIO Company, 2023

- monitoring of vibration values incl. frequency bands
- determine max velocity and frequencay at maximum

Customized modifications: -
------------------------

History:
-------
V4.11.1	20-01-2026	Bacci,	customized for DP29, generated from VibMonEG 4.11.1

Instructions FOR use:
--------------------
Sensor 1: Generator horizontal
Sensor 2: Generator vetical
Sensor 3: Engine horizontal
Sensor 4: Engine vetical

Outstandings:
------------

*******************************************************************************)

PROGRAM _INIT

//	(*========= DETERMINE POSITION OF X20CM4810 MODULE ==========*)
//	(* ********************************************************* *)
//	(*	reset variables											 *)
//	(* ********************************************************* *)
//	memset(ADR(sLabelInfo),	 	0, SIZEOF(sLabelInfo));
//
//	(* ********************************************************* *)
//	(*	get information about configured modules				 *)
//	(* ********************************************************* *)
//	xDiagCreateInfo_CM4810.enable	:= TRUE;
//	xDiagCreateInfo_CM4810.infoKind	:= asdiagCONFIGURED;
//	xDiagCreateInfo_CM4810();
//
//	IF (xDiagCreateInfo_CM4810.status = 0) THEN
//		iIdent 		:= xDiagCreateInfo_CM4810.ident;
//		iNrEntries	:= xDiagCreateInfo_CM4810.nrEntries;
//	END_IF;
//
//	(* ********************************************************* *)
//	(*	get module type of configured modules in Physical		 *)
//	(* ********************************************************* *)
//	FOR iIndex := 0 TO iNrEntries - 1 DO
//		xDiagGetStrInfo_CM4810.enable		:= TRUE;
//		xDiagGetStrInfo_CM4810.ident		:= iIdent;
//		xDiagGetStrInfo_CM4810.index		:= iIndex;
//		xDiagGetStrInfo_CM4810.infoCode		:= asdiagCONFIG_MODULE;
//		xDiagGetStrInfo_CM4810.pBuffer		:= ADR(sLabelInfo);
//		xDiagGetStrInfo_CM4810.bufferLen	:= SIZEOF(sLabelInfo) - 1;
//		xDiagGetStrInfo_CM4810();
//
//		IF (xDiagGetStrInfo_CM4810.status = 0) THEN
//		(* ********************************************************* *)
//		(*	get path of X20CM4810 module							 *)
//		(* ********************************************************* *)
//			IF FIND(sLabelInfo, 'X20CM4810') <> 0 THEN
//				xDiagGetStrInfo_CM4810.infoCode		:= asdiagPATH;
//				xDiagGetStrInfo_CM4810.pBuffer		:= ADR(sAddrInfo);
//				xDiagGetStrInfo_CM4810.bufferLen	:= SIZEOF(sAddrInfo) - 1;
//				xDiagGetStrInfo_CM4810();
//
//				IF (xDiagGetStrInfo_CM4810.status = 0) THEN
//					sCM4810Addr	:=	sAddrInfo;
//				END_IF;
//			END_IF;
//		END_IF;
//	END_FOR;
//
//	(* ********************************************************* *)
//	(*	free ressources of AsIODiag								 *)
//	(* ********************************************************* *)
//	xDiagDisposeInfo_CM4810.enable := TRUE;
//	xDiagDisposeInfo_CM4810.ident  := iIdent;
//	xDiagDisposeInfo_CM4810();
//	(*===========================================================*)

//  Prevent compiler warninga
	xDiagCreateInfo_CM4810.enable := FALSE;
	xDiagGetStrInfo_CM4810.enable := FALSE;
	xDiagDisposeInfo_CM4810.enable := FALSE;
	sLabelInfo;
	sAddrInfo;
	iIndex;
	iIdent;
	iNrEntries;

//  PLC address of 2nd X20CM4810 vibration module
	sCM4810Addr := 'IF3.ST33.IF1.ST3';

	(* init setting for CM4810 FUB *)
	xCM4810.paramMain.pModulePath			  := ADR(sCM4810Addr); 								(* set path to module *)

	xCM4810.enable							  := TRUE; 											(* enable FUB *)
	xCM4810.paramBufferUpload.nrArrayElements := SIZEOF(rData_x_Axis)/SIZEOF(rData_x_Axis[0]);	(* the length of the rData_x_Axis and rData_y_Axis arrays must be the same *)
	xCM4810.paramBufferUpload.pArrayXaxis	  := ADR(rData_x_Axis);								(* load buffer address x axis array *)
	xCM4810.paramBufferUpload.pArrayYaxis	  := ADR(rData_y_Axis);								(* load buffer address y axis array *)

	xCM4810.paramBufferUpload.moduleBuffer:= 66;    (* define module buffer for upload *)
	//moduleBuffer  Buffer description                        Signal source             Channel number   Number of values   y-axis unit    x-axis unit
	//    9         Buffered time signal (amplitude)          Raw acceleration signal      1                8192                [mg]       [seconds]
	//   11         Buffered time signal (amplitude)          Raw acceleration signal      2                8192                [mg]       [seconds]
	//   13         Buffered time signal (amplitude)          Raw acceleration signal      3                8192                [mg]       [seconds]
	//   15         Buffered time signal (amplitude)          Raw acceleration signal      4                8192                [mg]       [seconds]
	//   25         Buffered time signal (amplitude)          Envelope monitoring          1                8192                [mg]       [seconds]
	//   27         Buffered time signal (amplitude)          Envelope monitoring          2                8192                [mg]       [seconds]
	//   29         Buffered time signal (amplitude)          Envelope monitoring          3                8192                [mg]       [seconds]
	//   31         Buffered time signal (amplitude)          Envelope monitoring          4                8192                [mg]       [seconds]
	//   66         Spectrum buffered frequency (amplitude)   Raw velocity signal          1                4096                [mm/s]       [Hz]
	//   67         Spectrum buffered frequency (amplitude)   Raw acceleration signal      1                4096                [mg]         [Hz]
	//   70         Spectrum buffered frequency (amplitude)   Raw velocity signal          2                4096                [mm/s]       [Hz]
	//   71         Spectrum buffered frequency (amplitude)   Raw acceleration signal      2                4096                [mg]         [Hz]
	//   74         Spectrum buffered frequency (amplitude)   Raw velocity signal          3                4096                [mm/s]       [Hz]
	//   75         Spectrum buffered frequency (amplitude)   Raw acceleration signal      3                4096                [mg]         [Hz]
	//   78         Spectrum buffered frequency (amplitude)   Raw velocity signal          4                4096                [mm/s]       [Hz]
	//   79         Spectrum buffered frequency (amplitude)   Raw acceleration signal      4                4096                [mg]         [Hz]
	//   82         Spectrum buffered frequency (amplitude)   Envelope signal speed        1                4096                [mm/s]       [Hz]
	//   83         Spectrum buffered frequency (amplitude)   Envelope monitoring          1                4096                [mg]         [Hz]
	//   86         Spectrum buffered frequency (amplitude)   Envelope signal speed        2                4096                [mm/s]       [Hz]
	//   87         Spectrum buffered frequency (amplitude)   Envelope monitoring          2                4096                [mg]         [Hz]
	//   90         Spectrum buffered frequency (amplitude)   Envelope signal speed        3                4096                [mm/s]       [Hz]
	//   91         Spectrum buffered frequency (amplitude)   Envelope monitoring          3                4096                [mg]         [Hz]
	//   94         Spectrum buffered frequency (amplitude)   Envelope signal speed        4                4096                [mm/s]       [Hz]
	//   95         Spectrum buffered frequency (amplitude)   Envelope monitoring          4                4096                [mg]         [Hz]

	(* set sensor sensitivity *)
	rSensitivitySensor[1] := 100.0; (*mV/g*)
	rSensitivitySensor[2] := 100.0; (*mV/g*)
	rSensitivitySensor[3] := 100.0; (*mV/g*)
	rSensitivitySensor[4] := 100.0; (*mV/g*)

	(* Enable application of sensitivity on buffer *)
	xCM4810.paramMain.sensitivitySensor01:=rSensitivitySensor[1];
	xCM4810.paramMain.sensitivitySensor02:=rSensitivitySensor[2];
	xCM4810.paramMain.sensitivitySensor03:=rSensitivitySensor[3];
	xCM4810.paramMain.sensitivitySensor04:=rSensitivitySensor[4];

	(* initialize values *)
	tiCM4810_ReadBuffer := T#1m;
	iNum_VibSens		:= 1;

END_PROGRAM
```

#### VibMonEG.typ - Local data types
```iecst
TYPE
	stpCM4810_Enum :
		(
		stpInitDone,
		stpWaitStart,
		stpReqLockBuffer,
		stpUploadBuffer,
		stpReqUnlockBuffer,
		stpError
		);
END_TYPE
```

#### VibMonEG.var - Local variables
```iecst
VAR CONSTANT
	AxisArrayMaxIndex : UINT := 8191;
END_VAR
VAR
	bStartBufferUpload : BOOL := TRUE; (* in order to start the buffer upload, set to TRUE *)
	xCM4810 : vbioCtrlCM4810; (* FUB to read buffers of a CM4810 module *)
	stpCM4810 : stpCM4810_Enum; (* step of state machine *)
	rData_x_Axis : ARRAY[0..AxisArrayMaxIndex] OF REAL; (* array of x-axis values (time values [s] or frequency values [Hz]) *)
	rData_y_Axis : ARRAY[0..AxisArrayMaxIndex] OF REAL; (* array of y-axis values (vibration [mg] of [mm/s] values *)
	bWrite : BOOL;
	szWriteConfig : STRING[50];
	bRead : BOOL;
	szReadConfig : STRING[50];
	xAsIOAccWrite1 : AsIOAccWrite;
	xAsIOAccRead1 : AsIOAccRead;
	rSensitivitySensor : ARRAY[0..4] OF REAL;
	bGetFrequencyMax : BOOL;
	usCount : UINT;
	tiCM4810_ReadBuffer : TIME;
	xTON_ReadCycle : TON;
	iNum_VibSens : INT;
	rVel_VibSens_Band : ARRAY[0..32] OF REAL := [33(0)];
	rVel_VibSens : ARRAY[0..4] OF REAL := [5(0)];
	usMaxIndex : UINT;
	rVel_y_Axis_Max : REAL;
	bVibSens_Overflow : ARRAY[0..4] OF BOOL := [5(0)];
	bVibSens_BrokenWire : ARRAY[0..4] OF BOOL := [5(0)];
	ucWriteBandCnt : USINT := 0;
	rCenterBandOld1 : REAL := 0.0;
	rCenterBandOld2 : REAL := 0.0;
	rCenterBandOld3 : REAL := 0.0;
	rCenterBandOld4 : REAL := 0.0;
	rCenterBandOld5 : REAL := 0.0;
	rCenterBandOld6 : REAL := 0.0;
	rCenterBandOld7 : REAL := 0.0;
	rCenterBandOld8 : REAL := 0.0;
	rIdx_VibSens_BandWidtOld : REAL := 0.0;
END_VAR
VAR
	xDiagCreateInfo_CM4810 : DiagCreateInfo; (*Get number of configured modules*)
	xDiagGetStrInfo_CM4810 : DiagGetStrInfo; (*Get name of configured modules*)
	xDiagDisposeInfo_CM4810 : DiagDisposeInfo; (*Free ressources of AsIODiag*)
	sLabelInfo : STRING[50]; (*Includes label of configured module*)
	sAddrInfo : STRING[50]; (*Includes address of configured module*)
	iIndex : UDINT; (*Index of actual read module*)
	iIdent : UDINT; (*Ident from xDiagCreateInfo_CM4810*)
	iNrEntries : UDINT; (*Number of configured modules from xDiagCreateInfo_CM4810*)
	sCM4810Addr : STRING[50]; (*CM4810 IF PLC address string*)
END_VAR
```

### Program Logical/EngineGeneral/VibMon3EG (IEC, version 4.11.1) - Vibration monitoring eng & gen

#### VibMonEGCyclic.st - Init, cyclic, exit code
```iecst
(*******************************************************************************
VibMonEG: Vigration monitoring engine / generator (cyclic)

This code is confidential AND proprietary to the INNIO Company.
It may NOT be used in any form, or reproduced in any manner, without the express
written permission of the INNIO Company.
Copyright, INNIO Company, 2021

- monitoring of vibration values incl. frequency bands
- determine max velocity and frequencay at maximum

Customized modifications: -
------------------------

History:
-------
V4.11	25-05-2021	Weitzer, 	generated

Instructions FOR use:
--------------------
Sensor 1: Generator horizontal
Sensor 2: Generator vetical
Sensor 3: Engine horizontal
Sensor 4: Engine vetical

Outstandings:
------------

*******************************************************************************)

PROGRAM _CYCLIC

	(* code is only executed if function is activated by parameter and if system has completed the start up *)
	IF Para.bVibSens_Act AND IN_EG.tPB2MM.bSys_Run THEN

		(* mapping of data points from 4 vibration sensors *)
		FOR usCount := 0 TO 3 DO

			(* check if vibraton sensore wire break detected and engine speed is below start limit *)
			IF bVibSens_BrokenWire[usCount+1] OR IN_EG.rN_EngAct < Para.rN_EngStart_LimHi THEN
				(* vibration sensor live RMS values [mm/s]*)
				MM2VIS.rVel_VibSens[usCount+9] := 0;
				(* vibration sensor live frequency band [mm/s] *)
				MM2VIS.rVel_VibSens_Band1[usCount+9] := 0;
				MM2VIS.rVel_VibSens_Band2[usCount+9] := 0;
				MM2VIS.rVel_VibSens_Band3[usCount+9] := 0;
				MM2VIS.rVel_VibSens_Band4[usCount+9] := 0;
				MM2VIS.rVel_VibSens_Band5[usCount+9] := 0;
				MM2VIS.rVel_VibSens_Band6[usCount+9] := 0;
				MM2VIS.rVel_VibSens_Band7[usCount+9] := 0;
				MM2VIS.rVel_VibSens_Band8[usCount+9] := 0;
				(* vibration sensor max values *)
				MM2VIS.rVel_VibSens_Max[usCount+9] := 0;
				MM2VIS.rF_VibSens_Max[usCount+9]   := 0;
			(* check if no vibraton sensore overflow detected *)
			ELSIF NOT bVibSens_Overflow[usCount+1] THEN
				(* vibration sensor live RMS values [mm/s]*)
				MM2VIS.rVel_VibSens[usCount+9] := rVel_VibSens[usCount+1];					(* mapping directly from IO mapping, no HALIO used for vibration mesarurement *)
				(* vibration sensor live frequency band [mm/s] *)
				MM2VIS.rVel_VibSens_Band1[usCount+9] := rVel_VibSens_Band[usCount*8+1];		(* mapping directly from IO mapping, no HALIO used for vibration mesarurement *)
				MM2VIS.rVel_VibSens_Band2[usCount+9] := rVel_VibSens_Band[usCount*8+2];		(* mapping directly from IO mapping, no HALIO used for vibration mesarurement *)
				MM2VIS.rVel_VibSens_Band3[usCount+9] := rVel_VibSens_Band[usCount*8+3];		(* mapping directly from IO mapping, no HALIO used for vibration mesarurement *)
				MM2VIS.rVel_VibSens_Band4[usCount+9] := rVel_VibSens_Band[usCount*8+4];		(* mapping directly from IO mapping, no HALIO used for vibration mesarurement *)
				MM2VIS.rVel_VibSens_Band5[usCount+9] := rVel_VibSens_Band[usCount*8+5];		(* mapping directly from IO mapping, no HALIO used for vibration mesarurement *)
				MM2VIS.rVel_VibSens_Band6[usCount+9] := rVel_VibSens_Band[usCount*8+6];		(* mapping directly from IO mapping, no HALIO used for vibration mesarurement *)
				MM2VIS.rVel_VibSens_Band7[usCount+9] := rVel_VibSens_Band[usCount*8+7];		(* mapping directly from IO mapping, no HALIO used for vibration mesarurement *)
				MM2VIS.rVel_VibSens_Band8[usCount+9] := rVel_VibSens_Band[usCount*8+8];		(* mapping directly from IO mapping, no HALIO used for vibration mesarurement *)
			END_IF;

		END_FOR;

		(* read buffer data *)

		(* generate time interval for reading buffer *)
		xTON_ReadCycle(IN := NOT xTON_ReadCycle.Q, PT :=  tiCM4810_ReadBuffer);

		(* generate start reading trigger *)
		IF IN_EG.tEng_Run.Do AND stpCM4810 = stpWaitStart AND xTON_ReadCycle.Q THEN
			iNum_VibSens := iNum_VibSens + 1;
			IF iNum_VibSens > 4 THEN
				iNum_VibSens := 1;
			END_IF;
			bStartBufferUpload 					   := TRUE;
			xCM4810.paramBufferUpload.moduleBuffer := 66 + (iNum_VibSens-1) * 4;
		END_IF;

		(* state engine to read of data buffer *)

		CASE stpCM4810 OF
			//---------------------------------------------
			// wait for init done
			//---------------------------------------------
			stpInitDone:
				xCM4810.requestBufferLock := FALSE;
				xCM4810.uploadBuffer	  := FALSE;
				IF xCM4810.initDone AND xCM4810.moduleCfgUploadDone THEN
					stpCM4810 := stpWaitStart;
				END_IF;

			//---------------------------------------------
			// wait for start uplaod buffer
			//---------------------------------------------
			stpWaitStart:
				xCM4810.requestBufferLock := FALSE;
				xCM4810.uploadBuffer	  := FALSE;
				(* wait for start *)
				IF bStartBufferUpload THEN
					stpCM4810 := stpReqLockBuffer;
				END_IF;

			//---------------------------------------------
			// request lock buffer and wait until valid
			//---------------------------------------------
			stpReqLockBuffer:
				xCM4810.requestBufferLock := TRUE;
				bStartBufferUpload		  := FALSE; (* reset command start *)
				IF xCM4810.bufferLockValid THEN
					xCM4810.uploadBuffer := TRUE;
					stpCM4810			 := stpUploadBuffer;
				END_IF;

			//---------------------------------------------
			// upload buffer
			//---------------------------------------------
			stpUploadBuffer:
				IF xCM4810.bufferUploadDone THEN
					stpCM4810 := stpReqUnlockBuffer;
				END_IF;
				IF xCM4810.status <> ERR_FUB_BUSY AND xCM4810.status <> ERR_OK THEN
					stpCM4810 := stpError;
				END_IF

			//---------------------------------------------
			// unlock buffer and wait until valid
			//---------------------------------------------
			stpReqUnlockBuffer:
				xCM4810.requestBufferLock := FALSE;
				xCM4810.uploadBuffer	  := FALSE;
				IF NOT xCM4810.bufferLockValid THEN
					bGetFrequencyMax := TRUE;
					stpCM4810		 := stpWaitStart;
				END_IF;

			//---------------------------------------------
			// error
			//---------------------------------------------
			stpError:
			// no action!

		END_CASE;

		xCM4810.paramMain.pModulePath			  := ADR(sCM4810Addr);
		xCM4810.paramBufferUpload.pArrayXaxis	  := ADR(rData_x_Axis);
		xCM4810.paramBufferUpload.pArrayYaxis	  := ADR(rData_y_Axis);

		xCM4810(); (* call FUB exactly once per cycle *)

		(* get value & frequency max *)

		IF bGetFrequencyMax THEN

			MM2VIS.rF_VibSens_Max[iNum_VibSens+8]   := 0.0;		(* reset x(y max) max *)
			rVel_y_Axis_Max := 0.0;										(* reset y max *)
			usMaxIndex := 0;
			FOR usCount := 1 TO AxisArrayMaxIndex DO
				(* Upper limit for max value search at 500 Hz *)
				IF rData_x_Axis[usCount] > 500.0 THEN
					EXIT;
				END_IF
				(*find max signal value *)
				IF rData_y_Axis[usCount] > rVel_y_Axis_Max THEN
					rVel_y_Axis_Max := rData_y_Axis[usCount];		(* max virbration value *)
					MM2VIS.rF_VibSens_Max[iNum_VibSens+8]   := rData_x_Axis[usCount];		(* frequency at max virbration value *)
					usMaxIndex := usCount;
				END_IF
			END_FOR;

			(* correction of buffer value *)
			IF usMaxIndex > 1 AND usMaxIndex < (AxisArrayMaxIndex-2) THEN
				MM2VIS.rVel_VibSens_Max[iNum_VibSens+8] := 2.0/SQRT(3.0/2.0)*SQRT(0.5*(EXPT(rData_y_Axis[usMaxIndex-2],2)+EXPT(rData_y_Axis[usMaxIndex-1],2)+EXPT(rData_y_Axis[usMaxIndex],2)+EXPT(rData_y_Axis[usMaxIndex+1],2)+EXPT(rData_y_Axis[usMaxIndex+2],2)));
			ELSE
				MM2VIS.rVel_VibSens_Max[iNum_VibSens+8] := 0.0;
			END_IF;

			bGetFrequencyMax := FALSE;
		END_IF;

		(* calculate and display center frequency at the HMI *)

//		MM2VIS.rF_VibSens_CenterBand1 := Para.rN_EngNom/60.0*Para.rIdx_VibSens_BandOrder1;
//		MM2VIS.rF_VibSens_CenterBand2 := Para.rN_EngNom/60.0*Para.rIdx_VibSens_BandOrder2;
//		MM2VIS.rF_VibSens_CenterBand3 := Para.rN_EngNom/60.0*Para.rIdx_VibSens_BandOrder3;
//		MM2VIS.rF_VibSens_CenterBand4 := Para.rN_EngNom/60.0*Para.rIdx_VibSens_BandOrder4;
//		MM2VIS.rF_VibSens_CenterBand5 := Para.rN_EngNom/60.0*Para.rIdx_VibSens_BandOrder5;
//		MM2VIS.rF_VibSens_CenterBand6 := Para.rN_EngNom/60.0*Para.rIdx_VibSens_BandOrder6;
//		MM2VIS.rF_VibSens_CenterBand7 := Para.rN_EngNom/60.0*Para.rIdx_VibSens_BandOrder7;
//		MM2VIS.rF_VibSens_CenterBand8 := Para.rN_EngNom/60.0*Para.rIdx_VibSens_BandOrder8;

		(* check if band upper and lower frequency limit has to be set *)

		IF NOT bWrite THEN

			IF ucWriteBandCnt = 0 THEN

				IF Para.rIdx_VibSens_BandWidth <> rIdx_VibSens_BandWidtOld THEN
					rIdx_VibSens_BandWidtOld := Para.rIdx_VibSens_BandWidth;
					rCenterBandOld1			 := 0.0;
					rCenterBandOld2			 := 0.0;
					rCenterBandOld3			 := 0.0;
					rCenterBandOld4			 := 0.0;
					rCenterBandOld5			 := 0.0;
					rCenterBandOld6			 := 0.0;
					rCenterBandOld7			 := 0.0;
					rCenterBandOld8			 := 0.0;
				ELSIF MM2VIS.rF_VibSens_CenterBand1 <> rCenterBandOld1 THEN
					rCenterBandOld1 := MM2VIS.rF_VibSens_CenterBand1;
					ucWriteBandCnt  := 1;
				ELSIF MM2VIS.rF_VibSens_CenterBand2 <> rCenterBandOld2 THEN
					rCenterBandOld2 := MM2VIS.rF_VibSens_CenterBand2;
					ucWriteBandCnt  := 9;
				ELSIF MM2VIS.rF_VibSens_CenterBand3 <> rCenterBandOld3 THEN
					rCenterBandOld3 := MM2VIS.rF_VibSens_CenterBand3;
					ucWriteBandCnt  := 17;
				ELSIF MM2VIS.rF_VibSens_CenterBand4 <> rCenterBandOld4 THEN
					rCenterBandOld4 := MM2VIS.rF_VibSens_CenterBand4;
					ucWriteBandCnt  := 25;
				ELSIF MM2VIS.rF_VibSens_CenterBand5 <> rCenterBandOld5 THEN
					rCenterBandOld5 := MM2VIS.rF_VibSens_CenterBand5;
					ucWriteBandCnt  := 33;
				ELSIF MM2VIS.rF_VibSens_CenterBand6 <> rCenterBandOld6 THEN
					rCenterBandOld6 := MM2VIS.rF_VibSens_CenterBand6;
					ucWriteBandCnt  := 41;
				ELSIF MM2VIS.rF_VibSens_CenterBand7 <> rCenterBandOld7 THEN
					rCenterBandOld7 := MM2VIS.rF_VibSens_CenterBand7;
					ucWriteBandCnt  := 49;
				ELSIF MM2VIS.rF_VibSens_CenterBand8 <> rCenterBandOld8 THEN
					rCenterBandOld8 := MM2VIS.rF_VibSens_CenterBand8;
					ucWriteBandCnt  := 57;
				END_IF;

			END_IF;

			(* writing of the single band limit registers *)
			CASE ucWriteBandCnt OF

				(* Band 1 - Sensor 1 *)
				1:  bWrite		 		 := TRUE;
					szWriteConfig		 := 'FrequencyBand01LowerFrequency';
					xAsIOAccWrite1.value := LIMIT(1,REAL_TO_UDINT(4.0*(MM2VIS.rF_VibSens_CenterBand1 - Para.rIdx_VibSens_BandWidth/2)),40000);
					ucWriteBandCnt		 := 2;
				2:  bWrite		 		 := TRUE;
					szWriteConfig		 := 'FrequencyBand01UpperFrequency';
					xAsIOAccWrite1.value := LIMIT(1,REAL_TO_UDINT(4.0*(MM2VIS.rF_VibSens_CenterBand1 + Para.rIdx_VibSens_BandWidth/2)),40000);
					ucWriteBandCnt		 := 3;
				(* Band 1 - Sensor 2 *)
				3:  bWrite		 		 := TRUE;
					szWriteConfig		 := 'FrequencyBand09LowerFrequency';
					xAsIOAccWrite1.value := LIMIT(1,REAL_TO_UDINT(4.0*(MM2VIS.rF_VibSens_CenterBand1 - Para.rIdx_VibSens_BandWidth/2)),40000);
					ucWriteBandCnt		 := 4;
				4:  bWrite		 		 := TRUE;
					szWriteConfig		 := 'FrequencyBand09UpperFrequency';
					xAsIOAccWrite1.value := LIMIT(1,REAL_TO_UDINT(4.0*(MM2VIS.rF_VibSens_CenterBand1 + Para.rIdx_VibSens_BandWidth/2)),40000);
					ucWriteBandCnt		 := 5;
				(* Band 1 - Sensor 3 *)
				5:  bWrite		 		 := TRUE;
					szWriteConfig		 := 'FrequencyBand17LowerFrequency';
					xAsIOAccWrite1.value := LIMIT(1,REAL_TO_UDINT(4.0*(MM2VIS.rF_VibSens_CenterBand1 - Para.rIdx_VibSens_BandWidth/2)),40000);
					ucWriteBandCnt		 := 6;
				6:  bWrite		 		 := TRUE;
					szWriteConfig		 := 'FrequencyBand17UpperFrequency';
					xAsIOAccWrite1.value := LIMIT(1,REAL_TO_UDINT(4.0*(MM2VIS.rF_VibSens_CenterBand1 + Para.rIdx_VibSens_BandWidth/2)),40000);
					ucWriteBandCnt		 := 7;
				(* Band 1 - Sensor 4 *)
				7:  bWrite		 		 := TRUE;
					szWriteConfig		 := 'FrequencyBand25LowerFrequency';
					xAsIOAccWrite1.value := LIMIT(1,REAL_TO_UDINT(4.0*(MM2VIS.rF_VibSens_CenterBand1 - Para.rIdx_VibSens_BandWidth/2)),40000);
					ucWriteBandCnt		 := 8;
				8:  bWrite		 		 := TRUE;
					szWriteConfig		 := 'FrequencyBand25UpperFrequency';
					xAsIOAccWrite1.value := LIMIT(1,REAL_TO_UDINT(4.0*(MM2VIS.rF_VibSens_CenterBand1 + Para.rIdx_VibSens_BandWidth/2)),40000);
					ucWriteBandCnt		 := 0;

					(* Band 2 - Sensor 1 *)
				9:  bWrite		 		 := TRUE;
					szWriteConfig		 := 'FrequencyBand02LowerFrequency';
					xAsIOAccWrite1.value := LIMIT(1,REAL_TO_UDINT(4.0*(MM2VIS.rF_VibSens_CenterBand2 - Para.rIdx_VibSens_BandWidth/2)),40000);
					ucWriteBandCnt		 := 10;
				10: bWrite		 		 := TRUE;
					szWriteConfig		 := 'FrequencyBand02UpperFrequency';
					xAsIOAccWrite1.value := LIMIT(1,REAL_TO_UDINT(4.0*(MM2VIS.rF_VibSens_CenterBand2 + Para.rIdx_VibSens_BandWidth/2)),40000);
					ucWriteBandCnt		 := 11;
					(* Band 2 - Sensor 2 *)
				11: bWrite		 		 := TRUE;
					szWriteConfig		 := 'FrequencyBand10LowerFrequency';
					xAsIOAccWrite1.value := LIMIT(1,REAL_TO_UDINT(4.0*(MM2VIS.rF_VibSens_CenterBand2 - Para.rIdx_VibSens_BandWidth/2)),40000);
					ucWriteBandCnt		 := 12;
				12: bWrite		 		 := TRUE;
					szWriteConfig		 := 'FrequencyBand10UpperFrequency';
					xAsIOAccWrite1.value := LIMIT(1,REAL_TO_UDINT(4.0*(MM2VIS.rF_VibSens_CenterBand2 + Para.rIdx_VibSens_BandWidth/2)),40000);
					ucWriteBandCnt		 := 13;
					(* Band 2 - Sensor 3 *)
				13: bWrite		 		 := TRUE;
					szWriteConfig		 := 'FrequencyBand18LowerFrequency';
					xAsIOAccWrite1.value := LIMIT(1,REAL_TO_UDINT(4.0*(MM2VIS.rF_VibSens_CenterBand2 - Para.rIdx_VibSens_BandWidth/2)),40000);
					ucWriteBandCnt		 := 14;
				14: bWrite		 		 := TRUE;
					szWriteConfig		 := 'FrequencyBand18UpperFrequency';
					xAsIOAccWrite1.value := LIMIT(1,REAL_TO_UDINT(4.0*(MM2VIS.rF_VibSens_CenterBand2 + Para.rIdx_VibSens_BandWidth/2)),40000);
					ucWriteBandCnt		 := 15;
					(* Band 2 - Sensor 4 *)
				15: bWrite		 		 := TRUE;
					szWriteConfig		 := 'FrequencyBand26LowerFrequency';
					xAsIOAccWrite1.value := LIMIT(1,REAL_TO_UDINT(4.0*(MM2VIS.rF_VibSens_CenterBand2 - Para.rIdx_VibSens_BandWidth/2)),40000);
					ucWriteBandCnt		 := 16;
				16: bWrite		 		 := TRUE;
					szWriteConfig		 := 'FrequencyBand26UpperFrequency';
					xAsIOAccWrite1.value := LIMIT(1,REAL_TO_UDINT(4.0*(MM2VIS.rF_VibSens_CenterBand2 + Para.rIdx_VibSens_BandWidth/2)),40000);
					ucWriteBandCnt		 := 0;

					(* Band 3 - Sensor 1 *)
				17: bWrite		 		 := TRUE;
					szWriteConfig		 := 'FrequencyBand03LowerFrequency';
					xAsIOAccWrite1.value := LIMIT(1,REAL_TO_UDINT(4.0*(MM2VIS.rF_VibSens_CenterBand3 - Para.rIdx_VibSens_BandWidth/2)),40000);
					ucWriteBandCnt		 := 18;
				18: bWrite		 		 := TRUE;
					szWriteConfig		 := 'FrequencyBand03UpperFrequency';
					xAsIOAccWrite1.value := LIMIT(1,REAL_TO_UDINT(4.0*(MM2VIS.rF_VibSens_CenterBand3 + Para.rIdx_VibSens_BandWidth/2)),40000);
					ucWriteBandCnt		 := 19;
					(* Band 3 - Sensor 2 *)
				19: bWrite		 		 := TRUE;
					szWriteConfig		 := 'FrequencyBand11LowerFrequency';
					xAsIOAccWrite1.value := LIMIT(1,REAL_TO_UDINT(4.0*(MM2VIS.rF_VibSens_CenterBand3 - Para.rIdx_VibSens_BandWidth/2)),40000);
					ucWriteBandCnt		 := 20;
				20: bWrite		 		 := TRUE;
					szWriteConfig		 := 'FrequencyBand11UpperFrequency';
					xAsIOAccWrite1.value := LIMIT(1,REAL_TO_UDINT(4.0*(MM2VIS.rF_VibSens_CenterBand3 + Para.rIdx_VibSens_BandWidth/2)),40000);
					ucWriteBandCnt		 := 21;
					(* Band 3 - Sensor 3 *)
				21: bWrite		 		 := TRUE;
					szWriteConfig		 := 'FrequencyBand19LowerFrequency';
					xAsIOAccWrite1.value := LIMIT(1,REAL_TO_UDINT(4.0*(MM2VIS.rF_VibSens_CenterBand3 - Para.rIdx_VibSens_BandWidth/2)),40000);
					ucWriteBandCnt		 := 22;
				22: bWrite		 		 := TRUE;
					szWriteConfig		 := 'FrequencyBand19UpperFrequency';
					xAsIOAccWrite1.value := LIMIT(1,REAL_TO_UDINT(4.0*(MM2VIS.rF_VibSens_CenterBand3 + Para.rIdx_VibSens_BandWidth/2)),40000);
					ucWriteBandCnt		 := 23;
					(* Band 3 - Sensor 4 *)
				23: bWrite		 		 := TRUE;
					szWriteConfig		 := 'FrequencyBand27LowerFrequency';
					xAsIOAccWrite1.value := LIMIT(1,REAL_TO_UDINT(4.0*(MM2VIS.rF_VibSens_CenterBand3 - Para.rIdx_VibSens_BandWidth/2)),40000);
					ucWriteBandCnt		 := 24;
				24: bWrite		 		 := TRUE;
					szWriteConfig		 := 'FrequencyBand27UpperFrequency';
					xAsIOAccWrite1.value := LIMIT(1,REAL_TO_UDINT(4.0*(MM2VIS.rF_VibSens_CenterBand3 + Para.rIdx_VibSens_BandWidth/2)),40000);
					ucWriteBandCnt		 := 0;

					(* Band 4 - Sensor 1 *)
				25: bWrite		 		 := TRUE;
					szWriteConfig		 := 'FrequencyBand04LowerFrequency';
					xAsIOAccWrite1.value := LIMIT(1,REAL_TO_UDINT(4.0*(MM2VIS.rF_VibSens_CenterBand4 - Para.rIdx_VibSens_BandWidth/2)),40000);
					ucWriteBandCnt		 := 26;
				26: bWrite		 		 := TRUE;
					szWriteConfig		 := 'FrequencyBand04UpperFrequency';
					xAsIOAccWrite1.value := LIMIT(1,REAL_TO_UDINT(4.0*(MM2VIS.rF_VibSens_CenterBand4 + Para.rIdx_VibSens_BandWidth/2)),40000);
					ucWriteBandCnt		 := 27;
					(* Band 4 - Sensor 2 *)
				27: bWrite		 		 := TRUE;
					szWriteConfig		 := 'FrequencyBand12LowerFrequency';
					xAsIOAccWrite1.value := LIMIT(1,REAL_TO_UDINT(4.0*(MM2VIS.rF_VibSens_CenterBand4 - Para.rIdx_VibSens_BandWidth/2)),40000);
					ucWriteBandCnt		 := 28;
				28: bWrite		 		 := TRUE;
					szWriteConfig		 := 'FrequencyBand12UpperFrequency';
					xAsIOAccWrite1.value := LIMIT(1,REAL_TO_UDINT(4.0*(MM2VIS.rF_VibSens_CenterBand4 + Para.rIdx_VibSens_BandWidth/2)),40000);
					ucWriteBandCnt		 := 29;
					(* Band 4 - Sensor 3 *)
				29: bWrite		 		 := TRUE;
					szWriteConfig		 := 'FrequencyBand20LowerFrequency';
					xAsIOAccWrite1.value := LIMIT(1,REAL_TO_UDINT(4.0*(MM2VIS.rF_VibSens_CenterBand4 - Para.rIdx_VibSens_BandWidth/2)),40000);
					ucWriteBandCnt		 := 30;
				30: bWrite		 		 := TRUE;
					szWriteConfig		 := 'FrequencyBand20UpperFrequency';
					xAsIOAccWrite1.value := LIMIT(1,REAL_TO_UDINT(4.0*(MM2VIS.rF_VibSens_CenterBand4 + Para.rIdx_VibSens_BandWidth/2)),40000);
					ucWriteBandCnt		 := 31;
					(* Band 4 - Sensor 4 *)
				31: bWrite		 		 := TRUE;
					szWriteConfig		 := 'FrequencyBand28LowerFrequency';
					xAsIOAccWrite1.value := LIMIT(1,REAL_TO_UDINT(4.0*(MM2VIS.rF_VibSens_CenterBand4 - Para.rIdx_VibSens_BandWidth/2)),40000);
					ucWriteBandCnt		 := 32;
				32: bWrite		 		 := TRUE;
					szWriteConfig		 := 'FrequencyBand28UpperFrequency';
					xAsIOAccWrite1.value := LIMIT(1,REAL_TO_UDINT(4.0*(MM2VIS.rF_VibSens_CenterBand4 + Para.rIdx_VibSens_BandWidth/2)),40000);
					ucWriteBandCnt		 := 0;

					(* Band 5 - Sensor 1 *)
				33: bWrite		 		 := TRUE;
					szWriteConfig		 := 'FrequencyBand05LowerFrequency';
					xAsIOAccWrite1.value := LIMIT(1,REAL_TO_UDINT(4.0*(MM2VIS.rF_VibSens_CenterBand5 - Para.rIdx_VibSens_BandWidth/2)),40000);
					ucWriteBandCnt		 := 34;
				34: bWrite		 		 := TRUE;
					szWriteConfig		 := 'FrequencyBand05UpperFrequency';
					xAsIOAccWrite1.value := LIMIT(1,REAL_TO_UDINT(4.0*(MM2VIS.rF_VibSens_CenterBand5 + Para.rIdx_VibSens_BandWidth/2)),40000);
					ucWriteBandCnt		 := 35;
					(* Band 5 - Sensor 2 *)
				35: bWrite		 		 := TRUE;
					szWriteConfig		 := 'FrequencyBand13LowerFrequency';
					xAsIOAccWrite1.value := LIMIT(1,REAL_TO_UDINT(4.0*(MM2VIS.rF_VibSens_CenterBand5 - Para.rIdx_VibSens_BandWidth/2)),40000);
					ucWriteBandCnt		 := 36;
				36: bWrite		 		 := TRUE;
					szWriteConfig		 := 'FrequencyBand13UpperFrequency';
					xAsIOAccWrite1.value := LIMIT(1,REAL_TO_UDINT(4.0*(MM2VIS.rF_VibSens_CenterBand5 + Para.rIdx_VibSens_BandWidth/2)),40000);
					ucWriteBandCnt		 := 37;
					(* Band 5 - Sensor 3 *)
				37: bWrite		 		 := TRUE;
					szWriteConfig		 := 'FrequencyBand21LowerFrequency';
					xAsIOAccWrite1.value := LIMIT(1,REAL_TO_UDINT(4.0*(MM2VIS.rF_VibSens_CenterBand5 - Para.rIdx_VibSens_BandWidth/2)),40000);
					ucWriteBandCnt		 := 38;
				38: bWrite		 		 := TRUE;
					szWriteConfig		 := 'FrequencyBand21UpperFrequency';
					xAsIOAccWrite1.value := LIMIT(1,REAL_TO_UDINT(4.0*(MM2VIS.rF_VibSens_CenterBand5 + Para.rIdx_VibSens_BandWidth/2)),40000);
					ucWriteBandCnt		 := 39;
					(* Band 5 - Sensor 4 *)
				39: bWrite		 		 := TRUE;
					szWriteConfig		 := 'FrequencyBand29LowerFrequency';
					xAsIOAccWrite1.value := LIMIT(1,REAL_TO_UDINT(4.0*(MM2VIS.rF_VibSens_CenterBand5 - Para.rIdx_VibSens_BandWidth/2)),40000);
					ucWriteBandCnt		 := 40;
				40: bWrite		 		 := TRUE;
					szWriteConfig		 := 'FrequencyBand29UpperFrequency';
					xAsIOAccWrite1.value := LIMIT(1,REAL_TO_UDINT(4.0*(MM2VIS.rF_VibSens_CenterBand5 + Para.rIdx_VibSens_BandWidth/2)),40000);
					ucWriteBandCnt		 := 0;

					(* Band 6 - Sensor 1 *)
				41: bWrite		 		 := TRUE;
					szWriteConfig		 := 'FrequencyBand06LowerFrequency';
					xAsIOAccWrite1.value := LIMIT(1,REAL_TO_UDINT(4.0*(MM2VIS.rF_VibSens_CenterBand6 - Para.rIdx_VibSens_BandWidth/2)),40000);
					ucWriteBandCnt		 := 42;
				42: bWrite		 		 := TRUE;
					szWriteConfig		 := 'FrequencyBand06UpperFrequency';
					xAsIOAccWrite1.value := LIMIT(1,REAL_TO_UDINT(4.0*(MM2VIS.rF_VibSens_CenterBand6 + Para.rIdx_VibSens_BandWidth/2)),40000);
					ucWriteBandCnt		 := 43;
					(* Band 6 - Sensor 2 *)
				43: bWrite		 		 := TRUE;
					szWriteConfig		 := 'FrequencyBand14LowerFrequency';
					xAsIOAccWrite1.value := LIMIT(1,REAL_TO_UDINT(4.0*(MM2VIS.rF_VibSens_CenterBand6 - Para.rIdx_VibSens_BandWidth/2)),40000);
					ucWriteBandCnt		 := 44;
				44: bWrite		 		 := TRUE;
					szWriteConfig		 := 'FrequencyBand14UpperFrequency';
					xAsIOAccWrite1.value := LIMIT(1,REAL_TO_UDINT(4.0*(MM2VIS.rF_VibSens_CenterBand6 + Para.rIdx_VibSens_BandWidth/2)),40000);
					ucWriteBandCnt		 := 45;
					(* Band 6 - Sensor 3 *)
				45: bWrite		 		 := TRUE;
					szWriteConfig		 := 'FrequencyBand22LowerFrequency';
					xAsIOAccWrite1.value := LIMIT(1,REAL_TO_UDINT(4.0*(MM2VIS.rF_VibSens_CenterBand6 - Para.rIdx_VibSens_BandWidth/2)),40000);
					ucWriteBandCnt		 := 46;
				46: bWrite		 		 := TRUE;
					szWriteConfig		 := 'FrequencyBand22UpperFrequency';
					xAsIOAccWrite1.value := LIMIT(1,REAL_TO_UDINT(4.0*(MM2VIS.rF_VibSens_CenterBand6 + Para.rIdx_VibSens_BandWidth/2)),40000);
					ucWriteBandCnt		 := 47;
					(* Band 6 - Sensor 4 *)
				47: bWrite		 		 := TRUE;
					szWriteConfig		 := 'FrequencyBand30LowerFrequency';
					xAsIOAccWrite1.value := LIMIT(1,REAL_TO_UDINT(4.0*(MM2VIS.rF_VibSens_CenterBand6 - Para.rIdx_VibSens_BandWidth/2)),40000);
					ucWriteBandCnt		 := 48;
				48: bWrite		 		 := TRUE;
					szWriteConfig		 := 'FrequencyBand30UpperFrequency';
					xAsIOAccWrite1.value := LIMIT(1,REAL_TO_UDINT(4.0*(MM2VIS.rF_VibSens_CenterBand6 + Para.rIdx_VibSens_BandWidth/2)),40000);
					ucWriteBandCnt		 := 0;

					(* Band 7 - Sensor 1 *)
				49: bWrite		 		 := TRUE;
					szWriteConfig		 := 'FrequencyBand07LowerFrequency';
					xAsIOAccWrite1.value := LIMIT(1,REAL_TO_UDINT(4.0*(MM2VIS.rF_VibSens_CenterBand7 - Para.rIdx_VibSens_BandWidth/2)),40000);
					ucWriteBandCnt		 := 50;
				50: bWrite		 		 := TRUE;
					szWriteConfig		 := 'FrequencyBand07UpperFrequency';
					xAsIOAccWrite1.value := LIMIT(1,REAL_TO_UDINT(4.0*(MM2VIS.rF_VibSens_CenterBand7 + Para.rIdx_VibSens_BandWidth/2)),40000);
					ucWriteBandCnt		 := 51;
					(* Band 7 - Sensor 2 *)
				51: bWrite		 		 := TRUE;
					szWriteConfig		 := 'FrequencyBand15LowerFrequency';
					xAsIOAccWrite1.value := LIMIT(1,REAL_TO_UDINT(4.0*(MM2VIS.rF_VibSens_CenterBand7 - Para.rIdx_VibSens_BandWidth/2)),40000);
					ucWriteBandCnt		 := 52;
				52: bWrite		 		 := TRUE;
					szWriteConfig		 := 'FrequencyBand15UpperFrequency';
					xAsIOAccWrite1.value := LIMIT(1,REAL_TO_UDINT(4.0*(MM2VIS.rF_VibSens_CenterBand7 + Para.rIdx_VibSens_BandWidth/2)),40000);
					ucWriteBandCnt		 := 53;
					(* Band 7 - Sensor 3 *)
				53: bWrite		 		 := TRUE;
					szWriteConfig		 := 'FrequencyBand23LowerFrequency';
					xAsIOAccWrite1.value := LIMIT(1,REAL_TO_UDINT(4.0*(MM2VIS.rF_VibSens_CenterBand7 - Para.rIdx_VibSens_BandWidth/2)),40000);
					ucWriteBandCnt		 := 54;
				54: bWrite		 		 := TRUE;
					szWriteConfig		 := 'FrequencyBand23UpperFrequency';
					xAsIOAccWrite1.value := LIMIT(1,REAL_TO_UDINT(4.0*(MM2VIS.rF_VibSens_CenterBand7 + Para.rIdx_VibSens_BandWidth/2)),40000);
					ucWriteBandCnt		 := 55;
					(* Band 7 - Sensor 4 *)
				55: bWrite		 		 := TRUE;
					szWriteConfig		 := 'FrequencyBand31LowerFrequency';
					xAsIOAccWrite1.value := LIMIT(1,REAL_TO_UDINT(4.0*(MM2VIS.rF_VibSens_CenterBand7 - Para.rIdx_VibSens_BandWidth/2)),40000);
					ucWriteBandCnt		 := 56;
				56: bWrite		 		 := TRUE;
					szWriteConfig		 := 'FrequencyBand31UpperFrequency';
					xAsIOAccWrite1.value := LIMIT(1,REAL_TO_UDINT(4.0*(MM2VIS.rF_VibSens_CenterBand7 + Para.rIdx_VibSens_BandWidth/2)),40000);
					ucWriteBandCnt		 := 0;

					(* Band 8 - Sensor 1 *)
				57: bWrite		 		 := TRUE;
					szWriteConfig		 := 'FrequencyBand08LowerFrequency';
					xAsIOAccWrite1.value := LIMIT(1,REAL_TO_UDINT(4.0*(MM2VIS.rF_VibSens_CenterBand8 - Para.rIdx_VibSens_BandWidth/2)),40000);
					ucWriteBandCnt		 := 58;
				58: bWrite		 		 := TRUE;
					szWriteConfig		 := 'FrequencyBand08UpperFrequency';
					xAsIOAccWrite1.value := LIMIT(1,REAL_TO_UDINT(4.0*(MM2VIS.rF_VibSens_CenterBand8 + Para.rIdx_VibSens_BandWidth/2)),40000);
					ucWriteBandCnt		 := 59;
					(* Band 8 - Sensor 2 *)
				59: bWrite		 		 := TRUE;
					szWriteConfig		 := 'FrequencyBand16LowerFrequency';
					xAsIOAccWrite1.value := LIMIT(1,REAL_TO_UDINT(4.0*(MM2VIS.rF_VibSens_CenterBand8 - Para.rIdx_VibSens_BandWidth/2)),40000);
					ucWriteBandCnt		 := 60;
				60: bWrite		 		 := TRUE;
					szWriteConfig		 := 'FrequencyBand16UpperFrequency';
					xAsIOAccWrite1.value := LIMIT(1,REAL_TO_UDINT(4.0*(MM2VIS.rF_VibSens_CenterBand8 + Para.rIdx_VibSens_BandWidth/2)),40000);
					ucWriteBandCnt		 := 61;
					(* Band 8 - Sensor 3 *)
				61: bWrite		 		 := TRUE;
					szWriteConfig		 := 'FrequencyBand24LowerFrequency';
					xAsIOAccWrite1.value := LIMIT(1,REAL_TO_UDINT(4.0*(MM2VIS.rF_VibSens_CenterBand8 - Para.rIdx_VibSens_BandWidth/2)),40000);
					ucWriteBandCnt		 := 62;
				62: bWrite		 		 := TRUE;
					szWriteConfig		 := 'FrequencyBand24UpperFrequency';
					xAsIOAccWrite1.value := LIMIT(1,REAL_TO_UDINT(4.0*(MM2VIS.rF_VibSens_CenterBand8 + Para.rIdx_VibSens_BandWidth/2)),40000);
					ucWriteBandCnt		 := 63;
					(* Band 8 - Sensor 4 *)
				63: bWrite		 		 := TRUE;
					szWriteConfig		 := 'FrequencyBand32LowerFrequency';
					xAsIOAccWrite1.value := LIMIT(1,REAL_TO_UDINT(4.0*(MM2VIS.rF_VibSens_CenterBand8 - Para.rIdx_VibSens_BandWidth/2)),40000);
					ucWriteBandCnt		 := 64;
				64: bWrite		 		 := TRUE;
					szWriteConfig		 := 'FrequencyBand32UpperFrequency';
					xAsIOAccWrite1.value := LIMIT(1,REAL_TO_UDINT(4.0*(MM2VIS.rF_VibSens_CenterBand8 + Para.rIdx_VibSens_BandWidth/2)),40000);
					ucWriteBandCnt		 := 0;

			END_CASE;

		END_IF;

		(* read & write X204810 registers *)

		(* write band configuration and miscellaneous values *)
		IF bWrite THEN														(* set bWrite to TRUE to write a register on the CM48810 X20 module *)
			xAsIOAccWrite1.enable	    := TRUE;
			xAsIOAccWrite1.pDeviceName  := xCM4810.paramMain.pModulePath;
//			xAsIOAccWrite1.value	    := 0;								(* set value to write at this attribute of the function block *)
			xAsIOAccWrite1.pChannelName	:= ADR(szWriteConfig);				(* set name of register to write at string pv szWriteConfig *)
			xAsIOAccWrite1();

			IF xAsIOAccWrite1.status = 0 THEN
				bWrite := FALSE;
			END_IF;
		END_IF;

		(* read miscellaneous values *)
		IF bRead THEN														(* set bRead to TRUE to read a register from the CM48810 X20 module *)
			xAsIOAccRead1.enable	   := TRUE;
			xAsIOAccRead1.pDeviceName  := xCM4810.paramMain.pModulePath;
//			xAsIOAccRead1.value;											(* here the read valure can be found *)
			xAsIOAccRead1.pChannelName := ADR(szReadConfig);				(* set name of register to read at string pv szReadConfig *)
			xAsIOAccRead1();

			IF xAsIOAccRead1.status = 0 THEN
				bRead := FALSE;
			END_IF;
		END_IF;

	END_IF;

END_PROGRAM
```

#### VibMonEGInit.st
```iecst
(*******************************************************************************
VibMonEG: Vigration monitoring engine / generator (init)

This code is confidential AND proprietary to the INNIO Company.
It may NOT be used in any form, or reproduced in any manner, without the express
written permission of the INNIO Company.
Copyright, INNIO Company, 2023

- monitoring of vibration values incl. frequency bands
- determine max velocity and frequencay at maximum

Customized modifications: -
------------------------

History:
-------
V4.11.1	20-01-2026	Bacci,	customized for DP29, generated from VibMonEG 4.11.1

Instructions FOR use:
--------------------
Sensor 1: Generator horizontal
Sensor 2: Generator vetical
Sensor 3: Engine horizontal
Sensor 4: Engine vetical

Outstandings:
------------

*******************************************************************************)

PROGRAM _INIT

//	(*========= DETERMINE POSITION OF X20CM4810 MODULE ==========*)
//	(* ********************************************************* *)
//	(*	reset variables											 *)
//	(* ********************************************************* *)
//	memset(ADR(sLabelInfo),	 	0, SIZEOF(sLabelInfo));
//
//	(* ********************************************************* *)
//	(*	get information about configured modules				 *)
//	(* ********************************************************* *)
//	xDiagCreateInfo_CM4810.enable	:= TRUE;
//	xDiagCreateInfo_CM4810.infoKind	:= asdiagCONFIGURED;
//	xDiagCreateInfo_CM4810();
//
//	IF (xDiagCreateInfo_CM4810.status = 0) THEN
//		iIdent 		:= xDiagCreateInfo_CM4810.ident;
//		iNrEntries	:= xDiagCreateInfo_CM4810.nrEntries;
//	END_IF;
//
//	(* ********************************************************* *)
//	(*	get module type of configured modules in Physical		 *)
//	(* ********************************************************* *)
//	FOR iIndex := 0 TO iNrEntries - 1 DO
//		xDiagGetStrInfo_CM4810.enable		:= TRUE;
//		xDiagGetStrInfo_CM4810.ident		:= iIdent;
//		xDiagGetStrInfo_CM4810.index		:= iIndex;
//		xDiagGetStrInfo_CM4810.infoCode		:= asdiagCONFIG_MODULE;
//		xDiagGetStrInfo_CM4810.pBuffer		:= ADR(sLabelInfo);
//		xDiagGetStrInfo_CM4810.bufferLen	:= SIZEOF(sLabelInfo) - 1;
//		xDiagGetStrInfo_CM4810();
//
//		IF (xDiagGetStrInfo_CM4810.status = 0) THEN
//		(* ********************************************************* *)
//		(*	get path of X20CM4810 module							 *)
//		(* ********************************************************* *)
//			IF FIND(sLabelInfo, 'X20CM4810') <> 0 THEN
//				xDiagGetStrInfo_CM4810.infoCode		:= asdiagPATH;
//				xDiagGetStrInfo_CM4810.pBuffer		:= ADR(sAddrInfo);
//				xDiagGetStrInfo_CM4810.bufferLen	:= SIZEOF(sAddrInfo) - 1;
//				xDiagGetStrInfo_CM4810();
//
//				IF (xDiagGetStrInfo_CM4810.status = 0) THEN
//					sCM4810Addr	:=	sAddrInfo;
//				END_IF;
//			END_IF;
//		END_IF;
//	END_FOR;
//
//	(* ********************************************************* *)
//	(*	free ressources of AsIODiag								 *)
//	(* ********************************************************* *)
//	xDiagDisposeInfo_CM4810.enable := TRUE;
//	xDiagDisposeInfo_CM4810.ident  := iIdent;
//	xDiagDisposeInfo_CM4810();
//	(*===========================================================*)

//  Prevent compiler warninga
	xDiagCreateInfo_CM4810.enable := FALSE;
	xDiagGetStrInfo_CM4810.enable := FALSE;
	xDiagDisposeInfo_CM4810.enable := FALSE;
	sLabelInfo;
	sAddrInfo;
	iIndex;
	iIdent;
	iNrEntries;

//  PLC address of 3rd X20CM4810 vibration module
	sCM4810Addr := 'IF3.ST33.IF1.ST4';

	(* init setting for CM4810 FUB *)
	xCM4810.paramMain.pModulePath			  := ADR(sCM4810Addr); 								(* set path to module *)

	xCM4810.enable							  := TRUE; 											(* enable FUB *)
	xCM4810.paramBufferUpload.nrArrayElements := SIZEOF(rData_x_Axis)/SIZEOF(rData_x_Axis[0]);	(* the length of the rData_x_Axis and rData_y_Axis arrays must be the same *)
	xCM4810.paramBufferUpload.pArrayXaxis	  := ADR(rData_x_Axis);								(* load buffer address x axis array *)
	xCM4810.paramBufferUpload.pArrayYaxis	  := ADR(rData_y_Axis);								(* load buffer address y axis array *)

	xCM4810.paramBufferUpload.moduleBuffer:= 66;    (* define module buffer for upload *)
	//moduleBuffer  Buffer description                        Signal source             Channel number   Number of values   y-axis unit    x-axis unit
	//    9         Buffered time signal (amplitude)          Raw acceleration signal      1                8192                [mg]       [seconds]
	//   11         Buffered time signal (amplitude)          Raw acceleration signal      2                8192                [mg]       [seconds]
	//   13         Buffered time signal (amplitude)          Raw acceleration signal      3                8192                [mg]       [seconds]
	//   15         Buffered time signal (amplitude)          Raw acceleration signal      4                8192                [mg]       [seconds]
	//   25         Buffered time signal (amplitude)          Envelope monitoring          1                8192                [mg]       [seconds]
	//   27         Buffered time signal (amplitude)          Envelope monitoring          2                8192                [mg]       [seconds]
	//   29         Buffered time signal (amplitude)          Envelope monitoring          3                8192                [mg]       [seconds]
	//   31         Buffered time signal (amplitude)          Envelope monitoring          4                8192                [mg]       [seconds]
	//   66         Spectrum buffered frequency (amplitude)   Raw velocity signal          1                4096                [mm/s]       [Hz]
	//   67         Spectrum buffered frequency (amplitude)   Raw acceleration signal      1                4096                [mg]         [Hz]
	//   70         Spectrum buffered frequency (amplitude)   Raw velocity signal          2                4096                [mm/s]       [Hz]
	//   71         Spectrum buffered frequency (amplitude)   Raw acceleration signal      2                4096                [mg]         [Hz]
	//   74         Spectrum buffered frequency (amplitude)   Raw velocity signal          3                4096                [mm/s]       [Hz]
	//   75         Spectrum buffered frequency (amplitude)   Raw acceleration signal      3                4096                [mg]         [Hz]
	//   78         Spectrum buffered frequency (amplitude)   Raw velocity signal          4                4096                [mm/s]       [Hz]
	//   79         Spectrum buffered frequency (amplitude)   Raw acceleration signal      4                4096                [mg]         [Hz]
	//   82         Spectrum buffered frequency (amplitude)   Envelope signal speed        1                4096                [mm/s]       [Hz]
	//   83         Spectrum buffered frequency (amplitude)   Envelope monitoring          1                4096                [mg]         [Hz]
	//   86         Spectrum buffered frequency (amplitude)   Envelope signal speed        2                4096                [mm/s]       [Hz]
	//   87         Spectrum buffered frequency (amplitude)   Envelope monitoring          2                4096                [mg]         [Hz]
	//   90         Spectrum buffered frequency (amplitude)   Envelope signal speed        3                4096                [mm/s]       [Hz]
	//   91         Spectrum buffered frequency (amplitude)   Envelope monitoring          3                4096                [mg]         [Hz]
	//   94         Spectrum buffered frequency (amplitude)   Envelope signal speed        4                4096                [mm/s]       [Hz]
	//   95         Spectrum buffered frequency (amplitude)   Envelope monitoring          4                4096                [mg]         [Hz]

	(* set sensor sensitivity *)
	rSensitivitySensor[1] := 100.0; (*mV/g*)
	rSensitivitySensor[2] := 100.0; (*mV/g*)
	rSensitivitySensor[3] := 100.0; (*mV/g*)
	rSensitivitySensor[4] := 100.0; (*mV/g*)

	(* Enable application of sensitivity on buffer *)
	xCM4810.paramMain.sensitivitySensor01:=rSensitivitySensor[1];
	xCM4810.paramMain.sensitivitySensor02:=rSensitivitySensor[2];
	xCM4810.paramMain.sensitivitySensor03:=rSensitivitySensor[3];
	xCM4810.paramMain.sensitivitySensor04:=rSensitivitySensor[4];

	(* initialize values *)
	tiCM4810_ReadBuffer := T#1m;
	iNum_VibSens		:= 1;

END_PROGRAM
```

#### VibMonEG.typ - Local data types
```iecst
TYPE
	stpCM4810_Enum :
		(
		stpInitDone,
		stpWaitStart,
		stpReqLockBuffer,
		stpUploadBuffer,
		stpReqUnlockBuffer,
		stpError
		);
END_TYPE
```

#### VibMonEG.var - Local variables
```iecst
VAR CONSTANT
	AxisArrayMaxIndex : UINT := 8191;
END_VAR
VAR
	bStartBufferUpload : BOOL := TRUE; (* in order to start the buffer upload, set to TRUE *)
	xCM4810 : vbioCtrlCM4810; (* FUB to read buffers of a CM4810 module *)
	stpCM4810 : stpCM4810_Enum; (* step of state machine *)
	rData_x_Axis : ARRAY[0..AxisArrayMaxIndex] OF REAL; (* array of x-axis values (time values [s] or frequency values [Hz]) *)
	rData_y_Axis : ARRAY[0..AxisArrayMaxIndex] OF REAL; (* array of y-axis values (vibration [mg] of [mm/s] values *)
	bWrite : BOOL;
	szWriteConfig : STRING[50];
	bRead : BOOL;
	szReadConfig : STRING[50];
	xAsIOAccWrite1 : AsIOAccWrite;
	xAsIOAccRead1 : AsIOAccRead;
	rSensitivitySensor : ARRAY[0..4] OF REAL;
	bGetFrequencyMax : BOOL;
	usCount : UINT;
	tiCM4810_ReadBuffer : TIME;
	xTON_ReadCycle : TON;
	iNum_VibSens : INT;
	rVel_VibSens_Band : ARRAY[0..32] OF REAL := [33(0)];
	rVel_VibSens : ARRAY[0..4] OF REAL := [5(0)];
	usMaxIndex : UINT;
	rVel_y_Axis_Max : REAL;
	bVibSens_Overflow : ARRAY[0..4] OF BOOL := [5(0)];
	bVibSens_BrokenWire : ARRAY[0..4] OF BOOL := [5(0)];
	ucWriteBandCnt : USINT := 0;
	rCenterBandOld1 : REAL := 0.0;
	rCenterBandOld2 : REAL := 0.0;
	rCenterBandOld3 : REAL := 0.0;
	rCenterBandOld4 : REAL := 0.0;
	rCenterBandOld5 : REAL := 0.0;
	rCenterBandOld6 : REAL := 0.0;
	rCenterBandOld7 : REAL := 0.0;
	rCenterBandOld8 : REAL := 0.0;
	rIdx_VibSens_BandWidtOld : REAL := 0.0;
END_VAR
VAR
	xDiagCreateInfo_CM4810 : DiagCreateInfo; (*Get number of configured modules*)
	xDiagGetStrInfo_CM4810 : DiagGetStrInfo; (*Get name of configured modules*)
	xDiagDisposeInfo_CM4810 : DiagDisposeInfo; (*Free ressources of AsIODiag*)
	sLabelInfo : STRING[50]; (*Includes label of configured module*)
	sAddrInfo : STRING[50]; (*Includes address of configured module*)
	iIndex : UDINT; (*Index of actual read module*)
	iIdent : UDINT; (*Ident from xDiagCreateInfo_CM4810*)
	iNrEntries : UDINT; (*Number of configured modules from xDiagCreateInfo_CM4810*)
	sCM4810Addr : STRING[50]; (*CM4810 IF PLC address string*)
END_VAR
```

### Program Logical/EngineGeneral/PUscuffDet (IEC, version 4.11.0) - Power-unit scuffing detection

#### PUscuffDetCyclic.st - Cyclic code
```iecst
(********************************************************************************************************
PUscuffDet: 	crankcase pressure and knock noise signal based power-unit scuffing detection (cyclic)

This code is confidential AND proprietary TO the INNIO Company.
It may NOT be used in any form, or reproduced in any manner,
without written permission OF the INNIO Company.
Copyright, INNIO Company, 2022

Customized modifications:
------------------------

History:
-------
V4.11.00	14.01.2022	Schmidt		created

Outstandings:
------------
-
********************************************************************************************************)

PROGRAM _CYCLIC

	(* Parameters *)
	xPUscuff.Para.bPUscf_Ena 				:= Para.bPUscf_Ena AND xEngType.Type6 AND Para.bSA_KLS_Active;
	xPUscuff.Para.rTiPUscf_EnaDelay			:= Para.rTiPUscf_EnaDelay;
	xPUscuff.Para.rPUscf_Eps_scale			:= Para.rPUscf_Eps_scale;
	xPUscuff.Para.rTiPUscf_LearnReactDelay	:= Para.rTiPUscf_LearnReactDelay;
	xPUscuff.Para.rPr_CC_PUscf_Dev_HiHi		:= Para.rPr_CC_PUscf_Dev_HiHi*1000;
	xPUscuff.Para.rPUscf_LearnScale			:= Para.rPUscf_LearnScale;

	(* Inputs *)
	xPUscuff.In.bKnockSig 					:= IN_EG.bKnockSig;
	xPUscuff.In.rKnockNoise					:= IN_EG.rKnck_Noise;
	xPUscuff.In.iNumCyl						:= xEngType.NumberOfCylinder;
	xPUscuff.In.rP2s 						:= IN_EG.rPr_Ch_P2s_Avg;
	xPUscuff.In.rP_Act_Norm					:= IN_EG.rP_Act_Norm;
	xPUscuff.In.tPr_CC_Ai					:= (IN_EG.tPr_CC.Ai + rPr_CC_Ai_Offs)*1000;
	xPUscuff.In.tPr_CC_GoodQual				:= IN_EG.tPr_CC.GoodQual;
	xPUscuff.In.tGCB_On_Di 					:= IN_EG.tGCB_On.Di;
	xPUscuff.In.rKnockNoise					:= IN_EG.rKnck_Noise;

	(* Function execution *)
	xPUscuff();

	(* Outputs *)
	xPUscuff.Out.bPUscf_LearnEna;
	xPUscuff.Out.bPUscf_RelTrip;
	xPUscuff.Out.bPUscf_TripALL;
	xPUscuff.Out.bYpredict;
	xPUscuff.Out.rPr_CC_pred;
	xPUscuff.Out.tPUscuff_Map;

	(********************************************************************************************************************************)
	(************************              				 AMM sequencer	 		             	           **************************)
	(********************************************************************************************************************************)
	xTON_SecondTick(IN := NOT xTON_SecondTick.Q, PT:= T#800ms);					(* 800ms + 2x cycle time = 1 sec.*)

	(* Power-unit scuffing detection operating message *)
	xAmmSeq_PUscuff.Enable		:= NOT IN_EG.tAB2EG.bResetWarning;
	xAmmSeq_PUscuff.ClockPulse	:= xTON_SecondTick.Q;
	xAmmSeq_PUscuff.NrOfBits	:= 25;
	xAmmSeq_PUscuff.BitArray	:= ADR(xPUscuff.Out.bYpredict);
	xAmmSeq_PUscuff();

	bAMM_PUscuff				:= xPUscuff.Out.bPUscf_TripALL;
	bOpM_PUscuff				:= xAmmSeq_PUscuff.Alarm2;
	iNum_Msg2981				:= xAmmSeq_PUscuff.ErrorNr;

	(********************************************************************************************************************************)
	(************************              						VISU	 	             	   	        	*************************)
	(********************************************************************************************************************************)

	MM2VIS.iNum_Msg2981 	:= iNum_Msg2981;
	MM2VIS.bPUscf_RelTrip 	:= xPUscuff.Out.bPUscf_RelTrip;
	MM2VIS.bPUscf_LearnEna 	:= xPUscuff.Out.bPUscf_LearnEna;
	MM2VIS.rPr_CC_pred 		:= xPUscuff.Out.rPr_CC_pred;

END_PROGRAM
```

#### PUscuffDetInit.st - Init code
```iecst
(********************************************************************************************************
PUscuffDet: 	crankcase pressure and knock noise signal based power-unit scuffing detection (init)

This code is confidential AND proprietary TO the INNIO Company.
It may NOT be used in any form, or reproduced in any manner,
without written permission OF the INNIO Company.
Copyright, INNIO Company, 2022

Customized modifications:
------------------------

History:
-------
V4.11.00	14.01.2022	Schmidt		created

Outstandings:
------------
-
********************************************************************************************************)

PROGRAM _INIT

	xPUscuff(ssMethodType := 2);
	xPUscuff.ssMethodType := 3;

END_PROGRAM
```

#### PUscuffDet.var - Local variables
```iecst
VAR
	rPr_CC_Ai_Offs : REAL := 0.0; (*manual crankcase pressure offset*) (* *) (*V04.11.00.00*)
	xTON_SecondTick : TON := (0); (*FuB*) (* *) (*V04.11.00.00*)
	xAmmSeq_PUscuff : AmmSequence := (0); (*FuB*) (* *) (*V04.11.00.00*)
	iNum_Msg2981 : USINT := 0; (*PU scuffing - cylinder number*) (* *) (*V04.11.00.00*)
END_VAR
```

### Program Logical/EngineGeneral/Safety_PLC (IEC) - + Interface signals to/from SAFETY PLC

- Safety_PLCCyclic.st (not readable text: treated as protected, skipped)

- Safety_PLCInit.st (not readable text: treated as protected, skipped)

#### Safety_PLC.var
```iecst
VAR
	Data_sPLC : UDINT;
	i : UINT;
	szOptionNr : STRING[2];
	szSafeAppFilePath : STRING[260]; (*Filename of the SafeAPPLICATION file*)
	szSafeCommFilePath : STRING[260]; (*Filename of the SafeCOMMISSIONING file*)
	xEplSDORead : EplSDORead := (0);
	xSfDomainCompletion : SfDomainCompletion; (*Acknowledge the correctness of data on the SafeDOMAIN*)
	xSfDomainConnect : SfDomainConnect; (*Connects the specified user to the SafeDOMAIN *)
	xSfDomainControl : SfDomainControl; (*Execute predefined SafeDOMAIN actions*)
	xSfDomainExchange : SfDomainExchange; (*Confirm acknowledgment requests*)
	xSfDomainGetSafeNodeAvailability : SfDomainGetSafeNodeAvailability; (*Displays the value and attributes of a Safe node parameter *)
	xSfDomainGetSafeOptionBool : ARRAY[0..27] OF SfDomainGetSafeOptionBool; (*Displays the value and attributes of a Safe option BOOL parameter *)
	xSfDomainGetSafeOptionDint : ARRAY[0..27] OF SfDomainGetSafeOptionDint; (*Displays the value and attributes of a Safe option DINT  parameter *)
	xSfDomainInfo : SfDomainInfo; (*Read information from the SafeDOMAIN*)
	xSfDomainLoadSafeOptions : SfDomainLoadSafeOptions; (*Load the SafeCOMMISSIONING file for further processing*)
	xSfDomainSaveSafeOptions : SfDomainSaveSafeOptions; (*Saves the changed internal image of the SafeCOMMISSIONING file*)
	xSfDomainSetSafeNodeAvailability : SfDomainSetSafeNodeAvailability; (*Sets the value of the specified Safe node parameter *)
	xSfDomainSetSafeOptionBool : ARRAY[0..27] OF SfDomainSetSafeOptionBool; (*Sets the value of the specified Safe option BOOL parameter *)
	xSfDomainSetSafeOptionDint : ARRAY[0..27] OF SfDomainSetSafeOptionDint; (*Sets the value of the specified Safe option DINT parameter *)
	xCONV_HEX_CRC_Appl : CONV_HEX; (*FuB*)
	xCONV_HEX_CRC_ERV : CONV_HEX; (*FuB*)
	xCONV_HEX_CRC_HW : CONV_HEX; (*FuB*)
	xSfDomainTransfer : SfDomainTransfer; (*Transfer the SafeAPPLICATION and SafeCOMMISSIONING*)
END_VAR
```

### Package Logical/Exhaust - EX: Exhaust System

### Data object Logical/Exhaust/META_EX (Simple) - MODUL META data file
